// TwinCAT 3 PLC project TestHarnessCoreVerifier
// ProgramVersion: 3.1.4026.24
// libraries:
//   Tc2_Standard, * (Beckhoff Automation GmbH)
//   Tc2_System, * (Beckhoff Automation GmbH)
//   TestHarnessCore, * (None)
// project tree:
//   Doubles/ ConcurrencyWitness.TcPOU, ErroringTest.TcPOU, FailingTest.TcPOU, FakeTest.TcPOU, FakeTestWithAllHooks.TcPOU, FakeTestWithSetup.TcPOU, FloorTest.TcPOU, HangingBodyTest.TcPOU, HangingSetupTest.TcPOU, HangingTeardownTest.TcPOU, OrderedHooksTest.TcPOU, OrderWitness.TcPOU, PassingTest.TcPOU, RecordingReporter.TcPOU, SetupFailsTest.TcPOU, SlowSetupTest.TcPOU, SpanningTest.TcPOU, SpyReporter.TcPOU, StallingSuite.TcPOU, VerdictOnlyReporter.TcPOU, WitnessedTest.TcPOU
//   DUTs/ E_FloorStage.TcDUT, E_PureColour.TcDUT, ST_PureSample.TcDUT, ST_RecordedCase.TcDUT
//   Interfaces/ I_ProbeWitness.TcIO
//   / PlcTask.TcTTO
//   POUs/ MAIN.TcPOU, PRG_FloorCheck.TcPOU, PRG_UnitTests.TcPOU
//   Tests/Arbiter/ TEST_ArbiterAbandonEndsThePass.TcPOU, TEST_ArbiterCurrentIsNullWhenNothingActive.TcPOU, TEST_ArbiterEmptyPassIsComplete.TcPOU, TEST_ArbiterNotExhaustedWhileLastTestRuns.TcPOU, TEST_ArbiterRestartsFromTheBeginning.TcPOU, TEST_ArbiterVisitsEveryTestOnce.TcPOU
//   Tests/Assertions/ TEST_AssertBufferComparisons.TcPOU, TEST_AssertCompletedWithinCountsCompletedScans.TcPOU, TEST_AssertGreaterAndLessCompareTheRightWayRound.TcPOU, TEST_AssertInRangeIsInclusive.TcPOU, TEST_AssertNearUsesAbsoluteTolerance.TcPOU, TEST_AssertNotEqualRejectsSameness.TcPOU, TEST_AssertWithinUsesRelativeTolerance.TcPOU
//   Tests/Characterization/ CHAR_Capacity.TcPOU, CHAR_OverflowStatistics.TcPOU, CHAR_ReRunIndividual.TcPOU, CHAR_ReRunTests.TcPOU, CHAR_SerialExecution.TcPOU, CHAR_TimeoutPrecedence.TcPOU, CHAR_WallClockTimeout.TcPOU
//   Tests/EventReporter/ TEST_EventReporterDoesNotCallASkipAPass.TcPOU, TEST_EventReporterIsQuietAboutPasses.TcPOU, TEST_EventReporterNamesASkippedAndAnErroredRun.TcPOU, TEST_EventReporterRaisesEachOutcomeOnce.TcPOU, TEST_EventReporterSendsAndDoesNotFail.TcPOU, TEST_EventReporterWorksThroughTheFanout.TcPOU
//   Tests/Fanout/ TEST_FanoutCarriesTheSuiteResultThrough.TcPOU, TEST_FanoutForwardsRunStarted.TcPOU, TEST_FanoutIsIdleIsTheAndOfEverySink.TcPOU, TEST_FanoutNotifiesEverySinkInOrder.TcPOU, TEST_FanoutOnlyChecksGoToDetailSinks.TcPOU, TEST_FanoutRefusesBeyondCapacityAndTellsTheRest.TcPOU, TEST_FanoutSuspendSilencesEverything.TcPOU
//   Tests/Journal/ TEST_JournalDefaultsFillOnlyWhatWasNotClaimed.TcPOU, TEST_JournalResetKeepsWhatWasRegistered.TcPOU, TEST_JournalSkippedIsTerminalAndNotRed.TcPOU, TEST_JournalTimesOutOnCycles.TcPOU, TEST_JournalZeroBudgetDisablesTheDeadline.TcPOU
//   Tests/JUnitReporter/ TEST_JUnitReporterIsBusyWhileWriting.TcPOU, TEST_JUnitReporterOpensOnRunStarted.TcPOU, TEST_JUnitReporterRefusesWithNoPath.TcPOU, TEST_JUnitReporterReportsAFailedWrite.TcPOU, TEST_JUnitReporterWritesNothingWhenNothingRan.TcPOU, TEST_JUnitReporterWritesTheDocument.TcPOU
//   Tests/LogReporter/ TEST_LogReporterAlwaysWritesFrameworkErrors.TcPOU, TEST_LogReporterIsQuietAboutPasses.TcPOU, TEST_LogReporterNamesASkippedAndAnErroredRun.TcPOU, TEST_LogReporterNarratesSkipsOnlyWhenAsked.TcPOU, TEST_LogReporterNarratesWhenAsked.TcPOU, TEST_LogReporterSummarisesASuite.TcPOU, TEST_LogReporterWritesFailuresAndErrors.TcPOU
//   Tests/PureFunctions/ TEST_CompareNumericRules.TcPOU, TEST_CompareOtherRules.TcPOU, TEST_CompareTextRules.TcPOU, TEST_StopwatchMeasuresAndFreezes.TcPOU, TEST_SummaryLineComposition.TcPOU, TEST_ValueBriefShortens.TcPOU, TEST_ValueRendering.TcPOU
//   Tests/Registry/ TEST_RegistryCapacityAndOverflow.TcPOU, TEST_RegistryClosesRegistration.TcPOU, TEST_RegistryJournalRejectsBadIndex.TcPOU, TEST_RegistryJournalsArePerSlot.TcPOU, TEST_RegistryLookup.TcPOU, TEST_RegistryPreservesOrder.TcPOU, TEST_RegistryRejectsDuplicateLabel.TcPOU, TEST_RegistryRejectsEmptyLabelAndNullTest.TcPOU, TEST_RegistryResolvesOptionalHooks.TcPOU, TEST_RegistrySlotCarriesItsIndex.TcPOU
//   Tests/Runner/ TEST_RunnerAbandonMakesOneFinalCall.TcPOU, TEST_RunnerBodyDeadlineFires.TcPOU, TEST_RunnerDrivesThePhasesInOrder.TcPOU, TEST_RunnerRefusesAnEmptySlot.TcPOU, TEST_RunnerRunsAMultiScanBody.TcPOU, TEST_RunnerSetupDeadlineFires.TcPOU, TEST_RunnerSetupDoesNotSpendTheBodyBudget.TcPOU, TEST_RunnerSetupFailureSkipsTheBody.TcPOU, TEST_RunnerTeardownOverrunKeepsTheVerdict.TcPOU
//   Tests/Suite/ TEST_RegisteredAndReporterCountsAreReadable.TcPOU, TEST_RunAnnouncesItselfBeforeAnythingElse.TcPOU, TEST_RunOfOnlySkippedTestsIsSkipped.TcPOU, TEST_RunPassesWithSkipsBesideAPass.TcPOU, TEST_RunRefusingASuiteIsNeverSilent.TcPOU, TEST_RunReportsASkippedSuiteInItsPlace.TcPOU, TEST_RunReportsASuiteSkippedBeforeItsReporters.TcPOU, TEST_RunReportsEachSkippedTestByName.TcPOU, TEST_RunReRunDoesNotRunASkippedSuite.TcPOU, TEST_RunReRunReportsASkippedSuiteAgain.TcPOU, TEST_RunWithMoreSkipsThanPassesIsPassed.TcPOU, TEST_SuiteClosesRegistrationOnFirstEnable.TcPOU, TEST_SuiteDefaultsReachTheTests.TcPOU, TEST_SuiteRejectedRegistrationIsNeverSilent.TcPOU, TEST_SuiteReRunRepeatsTheRegisteredSet.TcPOU, TEST_SuiteReRunSingleRecordsNothing.TcPOU, TEST_SuiteRunsEveryRegisteredTest.TcPOU, TEST_SuiteSeparatesFailuresFromErrors.TcPOU, TEST_SuiteSkipMarksEverythingSkipped.TcPOU, TEST_SuiteSkippedAfterARejectedRegistrationIsErrored.TcPOU, TEST_SuiteSkippedWithNoLabelIsAFrameworkError.TcPOU, TEST_SuiteWithNoLabelIsAFrameworkError.TcPOU, TEST_SuiteWithNothingRegisteredIsComplete.TcPOU
//   Tests/Verdict/ TEST_VerdictFailIsAPlainFailure.TcPOU, TEST_VerdictFirstFailureWinsTheSummary.TcPOU, TEST_VerdictPassDoesNotOvertakeAFailure.TcPOU, TEST_VerdictRecordsAFailure.TcPOU, TEST_VerdictReportErrorIsNotAFailure.TcPOU, TEST_VerdictSummaryLeadsWithTheStepLabel.TcPOU, TEST_VerdictUntargetedHandleIsInert.TcPOU, TEST_VerdictZeroChecksIsErrored.TcPOU
//   Tests/Watchdog/ TEST_WatchdogAbandonsAStalledSuite.TcPOU, TEST_WatchdogMeasuresProgressNotTime.TcPOU, TEST_WatchdogZeroDisablesIt.TcPOU
// (motion and I/O tree: see PLC project testharnesscore)
// real-time tasks:
//   TASK PlcTask: cycle T#10ms, priority 20, ADS port 350

CONFIGURATION TestHarnessCoreVerifier
    RESOURCE PLC ON TwinCAT3
        TASK PlcTask(INTERVAL := T#10ms, PRIORITY := 20);
        PROGRAM MAIN WITH PlcTask : MAIN;
    END_RESOURCE
END_CONFIGURATION

// ---- DUTs/E_FloorStage.TcDUT
// Where the floor check has got to. One step per scan, so each stage's effect can

// be seen before the next runs.
{attribute 'qualified_only'}
{attribute 'strict'}
TYPE E_FloorStage : (
		Register := 0,
		Select	 := 1,
		Drive	 := 2,
		Read	 := 3,
		Done	 := 4
	) DINT;
END_TYPE

// ---- DUTs/E_PureColour.TcDUT
// A sample enum, for pinning that enums compare and render at all. The original

// rendered an unrecognised type class as an empty string, so a failed enum

// comparison read 'expected , actual ' - nothing, at the moment the reader most

// needed something.
{attribute 'qualified_only'}
TYPE E_PureColour : (
		Red	  := 0,
		Green := 1,
		Blue  := 2
	) DINT;
END_TYPE

// ---- DUTs/ST_PureSample.TcDUT
// A sample record for comparison tests. Shaped like a CoE object entry because

// that is the kind of struct a real test compares.
TYPE ST_PureSample :
	STRUCT
		Index	 : WORD;
		SubIndex : BYTE;
		Value	 : DINT;
	END_STRUCT
END_TYPE

// ---- DUTs/ST_RecordedCase.TcDUT
// One testcase as a recording sink captured it - the in-memory equivalent of a

// <testcase> node in the result document.

//

// The characterization tests ask questions of the ARTIFACT, not of the counters:

// how many cases, what failure type, does the message name the wall clock. This

// is what lets them, without a file to read back.
TYPE ST_RecordedCase :
	STRUCT
		Label	 : T_MaxString;
		Location : T_MaxString;
		Status	 : E_TestStatus;
		Kind	 : E_FailureKind;
		Summary	 : T_MaxString;
	END_STRUCT
END_TYPE

// ---- Interfaces/I_ProbeWitness.TcIO
// Somewhere for several spies to record the order they were notified in.

//

// An interface rather than a shared instance, because a spy holding the concrete

// type would be a second thing to keep wired up correctly.
INTERFACE I_ProbeWitness EXTENDS __SYSTEM.IQueryInterface

// Called by each spy as it is notified. Ordinal identifies which one.
METHOD Note
VAR_INPUT
	Ordinal : UDINT;
END_VAR
END_METHOD

END_INTERFACE

// ---- POUs/MAIN.TcPOU
// The verifier's task entry point.

//

// The floor check stands alone and runs first: it proves the harness can run a

// test at all, WITHOUT using the harness to prove it. Read PRG_FloorCheck.AllGood

// before trusting anything in PRG_UnitTests - if the runner is broken, every test

// reports NotStarted and that looks exactly like a wiring mistake.
PROGRAM MAIN

PRG_FloorCheck();
PRG_UnitTests();

END_PROGRAM

// ---- POUs/PRG_FloorCheck.TcPOU
// Proves the harness can run one test and report a verdict - WITHOUT using the

// harness to prove it.

//

// The verifier tests TestHarnessCore using TestHarnessCore. That is unavoidable

// and mostly fine, but it leaves one hole: if the runner never advances, every

// test reports NotStarted, and that looks exactly like a wiring mistake. There is

// no way to tell a framework defect from a setup error, because the thing

// reporting the result is the thing under test.

//

// So this drives TestRegistry, TestArbiter and TestRunner BY HAND, one step per

// scan, and writes what it finds into plain variables. Read them in the online

// view. Nothing between you and those objects is itself under test.

//

// EXPECTED once Stage reaches Done:

//

//   Claimed        TRUE          Advanced       TRUE

//   ActiveLabel    'floor'       Loaded         TRUE

//   Outcome        Finished      Verdict        Passed

//   Checks         1             BodyRunCount   1

//   Exhausted      TRUE          AllGood        TRUE

//

// AllGood is every line above, ANDed. If it is TRUE the floor holds, and any

// failure a real test reports afterwards is a real finding.

//

// If it is FALSE, read the values individually: the first wrong one names the

// object that broke.

//

// Re-run after ANY change to TestRunner, TestArbiter or TestRegistry. It costs one

// scan and it is the only check here that does not depend on what it tests.
PROGRAM PRG_FloorCheck
VAR
	// -- driven directly, not through a suite -----------------------------------
	Registry : TestRegistry<2>;
	Arbiter	 : TestArbiter;
	Runner	 : TestRunner;

	// The assertion handle. Named Handle, not Verdict, so it cannot be confused

	// with the verdict the test earns.
	Handle	: TestVerdict;
	Subject : FloorTest;
	Budgets : ST_TestBudgets;

	// -- what was found ---------------------------------------------------------
	Stage		 : E_FloorStage;
	Claimed		 : BOOL;
	Advanced	 : BOOL;
	ActiveLabel	 : T_MaxString;
	Loaded		 : BOOL;
	Outcome		 : E_PhaseOutcome;
	Verdict		 : E_TestStatus;
	Checks		 : UDINT;
	BodyRunCount : UDINT;
	Exhausted	 : BOOL;
	AllGood		 : BOOL;

	// -- working ----------------------------------------------------------------
	Slot	: ST_TestSlot;
	Journal : REFERENCE TO TestJournal;
	Fault	: E_RegistrationFault;
END_VAR

CASE Stage OF
	E_FloorStage.Register:
		// Capacity 2 holding one test. Capacity is not what is being checked here.
		Fault	:= Registry.TryClaim(Subject, 'floor', Budgets);
		Claimed := (Fault = E_RegistrationFault.None);
		Runner.Attach(Roster := Registry, Verdict := Handle);
		Arbiter.Attach(Registry);
		Arbiter.Begin();
		Stage := E_FloorStage.Select;

	E_FloorStage.Select:
		Advanced	:= Arbiter.Advance();
		Slot		:= Arbiter.Current;
		ActiveLabel := Slot.Label;
		Loaded		:= Runner.Load(Slot);
		Stage		:= E_FloorStage.Drive;

	E_FloorStage.Drive:
		// One scan of the body. A single-scan test must finish here; if it does not,
		// Outcome stays Running and that is itself the finding.
		Outcome := Runner.Advance(Enable := TRUE);
		IF Outcome <> E_PhaseOutcome.Running THEN
			Stage := E_FloorStage.Read;
		END_IF

	E_FloorStage.Read:
		Journal REF= Registry.Journal(0);
		IF __ISVALIDREF(Journal) THEN
			Verdict := Journal.Status;
			Checks	:= Journal.AssertionCount;
		END_IF

		BodyRunCount := Subject.RunCount;

		// Nothing left to hand out and nothing running.
		Arbiter.Advance();
		Exhausted := Arbiter.IsExhausted;
		AllGood	  := Claimed AND Advanced AND (ActiveLabel = 'floor') AND Loaded AND (Outcome = E_PhaseOutcome.Finished) AND (Verdict = E_TestStatus.Passed) AND (Checks = 1) AND (BodyRunCount = 1) AND Exhausted;
		Stage	  := E_FloorStage.Done;

	E_FloorStage.Done:
		// Terminal. Nothing repeats, so every value above stays readable.
		;
END_CASE

END_PROGRAM

// ---- Doubles/FloorTest.TcPOU
// The simplest thing that can be called a test: one check, finished in one scan.

//

// Nothing optional, nothing multi-scan, nothing that can fail. If the harness

// cannot run THIS and report Passed, no other result it produces means anything.
FUNCTION_BLOCK FloorTest IMPLEMENTS I_Test
VAR
	// Counted so the floor check can prove the body ran exactly once. A harness

	// that called it twice, or never, would otherwise look identical from outside.
	_RunCount : UDINT;
END_VAR

METHOD Run : BOOL
VAR_INPUT
	Enable : BOOL;
	Test   : I_TestAssertions;
END_VAR

VAR
	// AssertEqual takes ANY, which binds only to an addressable variable - a

	// literal or an inlined expression will not compile. Both sides are copied into

	// variables first. A language constraint, not a choice.
	Expected : DINT := 4;
	Actual	 : DINT;
	Two		 : DINT := 2;
END_VAR
IF NOT Enable THEN
	// Abandoned. Nothing to unwind.
	Run := TRUE;
	RETURN;
END_IF

_RunCount := _RunCount + 1;
Actual	  := Two + Two;
Test.AssertEqual(Expected, Actual, 'two and two');
Run := TRUE;
END_METHOD

// How many times the harness called Run. Exactly 1 after a clean single run.
PROPERTY RunCount : UDINT
GET
RunCount := _RunCount;
END_GET
END_PROPERTY

END_FUNCTION_BLOCK

// ---- POUs/PRG_UnitTests.TcPOU
// The composition root: what is registered, what reports it, and the run that
// drives it.
//
// This is also a WORKED EXAMPLE. It composes the library the way a real project
// should - a run, a suite, three sinks - so anything awkward here is awkward for
// everyone.
//
// READ THESE, in the online view:
//
//   Complete   TRUE once every test has finished
//   Outcome    Passed if the library is sound
//   Total      111 - assert this. A test that stops being registered vanishes
//              silently, and CI sees fewer passes rather than a failure
//   Passed / Failed / Errors / Skipped
//   Idle       TRUE once the result document has reached disk. CI MUST WAIT FOR
//              BOTH Complete AND Idle - a run finishing and its file landing are
//              different events, and copying between them yields a truncated
//              artifact that reads as a broken pipeline
//
// WHERE A FAILURE SHOWS UP:
//   - the Logged Events window, as a log line and as an event
//   - C:\ProgramData\Beckhoff\TwinCAT\3.1\Boot\TestHarnessCoreResults.xml
//
// Read the failure there rather than from journal internals in a watch window.
// Making that unnecessary is what this library is for.
//
// THE FAILURE PATH IS EXERCISED, not assumed. The Verdict tests drive DELIBERATE
// failures into a private journal; the Suite tests register doubles that fail and
// error on purpose; the JUnit tests write to a folder that does not exist. They all
// pass. What they prove is that going wrong works.
//
// THE CHARACTERIZATION TESTS ARE THE ACCEPTANCE CONTRACT - behaviour a project
// depending on this library is entitled to rely on. They are also the only tests
// that ask questions of the ARTIFACT: how many cases the document carries, what
// type attribute a failure got, whether a timeout message names the wall clock.
//
// MULTI-SCAN TESTS hold a private runner, suite or run and step it one scan per
// call, returning FALSE until it finishes - the same mechanism they are verifying,
// one level down. Each carries a watchdog, so a defect that never completes fails
// its own test rather than hanging everything and looking like a broken verifier.
PROGRAM PRG_UnitTests
VAR
	// A RUN, not just a suite. RunFinished is a run-level event and only a TestRun
	// raises it - which is what produces a document at all.
	Runner : TestRun<2>;
	Suite  : TestSuite<130>;

	// All three sinks, which is the realistic composition: a log line to read at a
	// glance, an event to filter and route, a document for CI.
	LogSink	  : TestLogReporter;
	EventSink : TestEventReporter;
	JUnitSink : TestJUnitReporter;

	// The 4026 boot folder. Named apart from the files the JUnit tests write, so a
	// stale artifact from either cannot be mistaken for the other.
	ResultPath : T_MaxString := 'C:\ProgramData\Beckhoff\TwinCAT\3.1\Boot\TestHarnessCoreResults.xml';

	Budgets : ST_TestBudgets;
	Wired	: BOOL;

	// -- Registry --
	registryCapacityAndOverflow	: TEST_RegistryCapacityAndOverflow;
	registryRejectsDuplicateLabel	: TEST_RegistryRejectsDuplicateLabel;
	registryRejectsEmptyLabelAndNullTest	: TEST_RegistryRejectsEmptyLabelAndNullTest;
	registryClosesRegistration	: TEST_RegistryClosesRegistration;
	registryLookup	: TEST_RegistryLookup;
	registryPreservesOrder	: TEST_RegistryPreservesOrder;
	registrySlotCarriesItsIndex	: TEST_RegistrySlotCarriesItsIndex;
	registryResolvesOptionalHooks	: TEST_RegistryResolvesOptionalHooks;
	registryJournalsArePerSlot	: TEST_RegistryJournalsArePerSlot;
	registryJournalRejectsBadIndex	: TEST_RegistryJournalRejectsBadIndex;

	// -- Arbiter --
	arbiterVisitsEveryTestOnce	: TEST_ArbiterVisitsEveryTestOnce;
	arbiterCurrentIsNullWhenNothingActive	: TEST_ArbiterCurrentIsNullWhenNothingActive;
	arbiterEmptyPassIsComplete	: TEST_ArbiterEmptyPassIsComplete;
	arbiterAbandonEndsThePass	: TEST_ArbiterAbandonEndsThePass;
	arbiterNotExhaustedWhileLastTestRuns	: TEST_ArbiterNotExhaustedWhileLastTestRuns;
	arbiterRestartsFromTheBeginning	: TEST_ArbiterRestartsFromTheBeginning;

	// -- Verdict --
	verdictRecordsAFailure	: TEST_VerdictRecordsAFailure;
	verdictPassDoesNotOvertakeAFailure	: TEST_VerdictPassDoesNotOvertakeAFailure;
	verdictZeroChecksIsErrored	: TEST_VerdictZeroChecksIsErrored;
	verdictReportErrorIsNotAFailure	: TEST_VerdictReportErrorIsNotAFailure;
	verdictFailIsAPlainFailure	: TEST_VerdictFailIsAPlainFailure;
	verdictSummaryLeadsWithTheStepLabel	: TEST_VerdictSummaryLeadsWithTheStepLabel;
	verdictFirstFailureWinsTheSummary	: TEST_VerdictFirstFailureWinsTheSummary;
	verdictUntargetedHandleIsInert	: TEST_VerdictUntargetedHandleIsInert;

	// -- Journal --
	journalTimesOutOnCycles	: TEST_JournalTimesOutOnCycles;
	journalZeroBudgetDisablesTheDeadline	: TEST_JournalZeroBudgetDisablesTheDeadline;
	journalDefaultsFillOnlyWhatWasNotClaimed	: TEST_JournalDefaultsFillOnlyWhatWasNotClaimed;
	journalResetKeepsWhatWasRegistered	: TEST_JournalResetKeepsWhatWasRegistered;
	journalSkippedIsTerminalAndNotRed	: TEST_JournalSkippedIsTerminalAndNotRed;

	// -- Runner --
	runnerDrivesThePhasesInOrder	: TEST_RunnerDrivesThePhasesInOrder;
	runnerRunsAMultiScanBody	: TEST_RunnerRunsAMultiScanBody;
	runnerSetupFailureSkipsTheBody	: TEST_RunnerSetupFailureSkipsTheBody;
	runnerSetupDoesNotSpendTheBodyBudget	: TEST_RunnerSetupDoesNotSpendTheBodyBudget;
	runnerBodyDeadlineFires	: TEST_RunnerBodyDeadlineFires;
	runnerSetupDeadlineFires	: TEST_RunnerSetupDeadlineFires;
	runnerTeardownOverrunKeepsTheVerdict	: TEST_RunnerTeardownOverrunKeepsTheVerdict;
	runnerAbandonMakesOneFinalCall	: TEST_RunnerAbandonMakesOneFinalCall;
	runnerRefusesAnEmptySlot	: TEST_RunnerRefusesAnEmptySlot;

	// -- Suite --
	suiteRunsEveryRegisteredTest	: TEST_SuiteRunsEveryRegisteredTest;
	suiteSeparatesFailuresFromErrors	: TEST_SuiteSeparatesFailuresFromErrors;
	suiteClosesRegistrationOnFirstEnable	: TEST_SuiteClosesRegistrationOnFirstEnable;
	suiteRejectedRegistrationIsNeverSilent	: TEST_SuiteRejectedRegistrationIsNeverSilent;
	suiteSkipMarksEverythingSkipped	: TEST_SuiteSkipMarksEverythingSkipped;
	suiteSkippedAfterARejectedRegistrationIsErrored	: TEST_SuiteSkippedAfterARejectedRegistrationIsErrored;
	suiteSkippedWithNoLabelIsAFrameworkError	: TEST_SuiteSkippedWithNoLabelIsAFrameworkError;
	suiteReRunRepeatsTheRegisteredSet	: TEST_SuiteReRunRepeatsTheRegisteredSet;
	suiteReRunSingleRecordsNothing	: TEST_SuiteReRunSingleRecordsNothing;
	suiteWithNothingRegisteredIsComplete	: TEST_SuiteWithNothingRegisteredIsComplete;
	suiteWithNoLabelIsAFrameworkError	: TEST_SuiteWithNoLabelIsAFrameworkError;
	suiteDefaultsReachTheTests	: TEST_SuiteDefaultsReachTheTests;

	runAnnouncesItselfBeforeAnythingElse	: TEST_RunAnnouncesItselfBeforeAnythingElse;
	runRefusingASuiteIsNeverSilent	: TEST_RunRefusingASuiteIsNeverSilent;
	runPassesWithSkipsBesideAPass	: TEST_RunPassesWithSkipsBesideAPass;
	runOfOnlySkippedTestsIsSkipped	: TEST_RunOfOnlySkippedTestsIsSkipped;
	runWithMoreSkipsThanPassesIsPassed	: TEST_RunWithMoreSkipsThanPassesIsPassed;
	runReportsASuiteSkippedBeforeItsReporters	: TEST_RunReportsASuiteSkippedBeforeItsReporters;
	runReportsASkippedSuiteInItsPlace	: TEST_RunReportsASkippedSuiteInItsPlace;
	runReportsEachSkippedTestByName	: TEST_RunReportsEachSkippedTestByName;
	runReRunDoesNotRunASkippedSuite	: TEST_RunReRunDoesNotRunASkippedSuite;
	runReRunReportsASkippedSuiteAgain	: TEST_RunReRunReportsASkippedSuiteAgain;

	// -- Fanout --
	fanoutNotifiesEverySinkInOrder	: TEST_FanoutNotifiesEverySinkInOrder;
	fanoutOnlyChecksGoToDetailSinks	: TEST_FanoutOnlyChecksGoToDetailSinks;
	fanoutIsIdleIsTheAndOfEverySink	: TEST_FanoutIsIdleIsTheAndOfEverySink;
	fanoutSuspendSilencesEverything	: TEST_FanoutSuspendSilencesEverything;
	fanoutRefusesBeyondCapacityAndTellsTheRest	: TEST_FanoutRefusesBeyondCapacityAndTellsTheRest;
	fanoutCarriesTheSuiteResultThrough	: TEST_FanoutCarriesTheSuiteResultThrough;

	fanoutForwardsRunStarted	: TEST_FanoutForwardsRunStarted;

	// -- LogReporter --
	logReporterIsQuietAboutPasses	: TEST_LogReporterIsQuietAboutPasses;
	logReporterWritesFailuresAndErrors	: TEST_LogReporterWritesFailuresAndErrors;
	logReporterNarratesWhenAsked	: TEST_LogReporterNarratesWhenAsked;
	logReporterAlwaysWritesFrameworkErrors	: TEST_LogReporterAlwaysWritesFrameworkErrors;
	logReporterSummarisesASuite	: TEST_LogReporterSummarisesASuite;
	logReporterNarratesSkipsOnlyWhenAsked	: TEST_LogReporterNarratesSkipsOnlyWhenAsked;
	logReporterNamesASkippedAndAnErroredRun	: TEST_LogReporterNamesASkippedAndAnErroredRun;

	jUnitReporterOpensOnRunStarted	: TEST_JUnitReporterOpensOnRunStarted;

	// -- EventReporter --
	eventReporterSendsAndDoesNotFail	: TEST_EventReporterSendsAndDoesNotFail;
	eventReporterIsQuietAboutPasses	: TEST_EventReporterIsQuietAboutPasses;
	eventReporterRaisesEachOutcomeOnce	: TEST_EventReporterRaisesEachOutcomeOnce;
	eventReporterWorksThroughTheFanout	: TEST_EventReporterWorksThroughTheFanout;
	eventReporterDoesNotCallASkipAPass	: TEST_EventReporterDoesNotCallASkipAPass;
	eventReporterNamesASkippedAndAnErroredRun	: TEST_EventReporterNamesASkippedAndAnErroredRun;

	// -- JUnitReporter --
	jUnitReporterWritesTheDocument	: TEST_JUnitReporterWritesTheDocument;
	jUnitReporterIsBusyWhileWriting	: TEST_JUnitReporterIsBusyWhileWriting;
	jUnitReporterReportsAFailedWrite	: TEST_JUnitReporterReportsAFailedWrite;
	jUnitReporterRefusesWithNoPath	: TEST_JUnitReporterRefusesWithNoPath;
	jUnitReporterWritesNothingWhenNothingRan	: TEST_JUnitReporterWritesNothingWhenNothingRan;

	// -- Pure functions: the comparison and rendering rules --
	compareNumericRules	: TEST_CompareNumericRules;
	compareTextRules	: TEST_CompareTextRules;
	compareOtherRules	: TEST_CompareOtherRules;
	summaryLineComposition	: TEST_SummaryLineComposition;
	valueRendering	: TEST_ValueRendering;
	valueBriefShortens	: TEST_ValueBriefShortens;

	// -- Assertions: the public surface every user touches --
	assertNotEqualRejectsSameness	: TEST_AssertNotEqualRejectsSameness;
	assertGreaterAndLessCompareTheRightWayRound	: TEST_AssertGreaterAndLessCompareTheRightWayRound;
	assertNearUsesAbsoluteTolerance	: TEST_AssertNearUsesAbsoluteTolerance;
	assertWithinUsesRelativeTolerance	: TEST_AssertWithinUsesRelativeTolerance;
	assertInRangeIsInclusive	: TEST_AssertInRangeIsInclusive;
	assertBufferComparisons	: TEST_AssertBufferComparisons;
	assertCompletedWithinCountsCompletedScans	: TEST_AssertCompletedWithinCountsCompletedScans;

	stopwatchMeasuresAndFreezes	: TEST_StopwatchMeasuresAndFreezes;
	registeredAndReporterCountsAreReadable	: TEST_RegisteredAndReporterCountsAreReadable;
	// -- Suite watchdog --
	watchdogAbandonsAStalledSuite	: TEST_WatchdogAbandonsAStalledSuite;
	watchdogMeasuresProgressNotTime	: TEST_WatchdogMeasuresProgressNotTime;
	watchdogZeroDisablesIt	: TEST_WatchdogZeroDisablesIt;

	// -- Characterization: the acceptance contract --
	cHAR_Capacity	: CHAR_Capacity;
	cHAR_OverflowStatistics	: CHAR_OverflowStatistics;
	cHAR_ReRunTests	: CHAR_ReRunTests;
	cHAR_ReRunIndividual	: CHAR_ReRunIndividual;
	cHAR_WallClockTimeout	: CHAR_WallClockTimeout;
	cHAR_TimeoutPrecedence	: CHAR_TimeoutPrecedence;
	cHAR_SerialExecution	: CHAR_SerialExecution;

	// -- the result, for the watch window ---------------------------------------
	Complete : BOOL;
	Outcome	 : E_RunOutcome;
	Total	 : UDINT;
	Passed	 : UDINT;
	Failed	 : UDINT;
	Errors	 : UDINT;
	Skipped	 : UDINT;
	Duration : LREAL;

	// -- did the artifact land? -------------------------------------------------
	Idle		  : BOOL;
	FilesWritten  : UDINT;
	WriteFailures : UDINT;
END_VAR

IF NOT Wired THEN
	Wired := TRUE;

	Suite.SetLabel('TestHarnessCore');

	// Registry
	Suite.Register(registryCapacityAndOverflow, 'Registry: capacity and overflow', Budgets);
	Suite.Register(registryRejectsDuplicateLabel, 'Registry: rejects a duplicate label', Budgets);
	Suite.Register(registryRejectsEmptyLabelAndNullTest, 'Registry: rejects an empty label and a null test', Budgets);
	Suite.Register(registryClosesRegistration, 'Registry: closes registration on first enable', Budgets);
	Suite.Register(registryLookup, 'Registry: lookup by label', Budgets);
	Suite.Register(registryPreservesOrder, 'Registry: preserves registration order', Budgets);
	Suite.Register(registrySlotCarriesItsIndex, 'Registry: a slot carries its own index', Budgets);
	Suite.Register(registryResolvesOptionalHooks, 'Registry: resolves the optional hooks independently', Budgets);
	Suite.Register(registryJournalsArePerSlot, 'Registry: journals are per slot and live', Budgets);
	Suite.Register(registryJournalRejectsBadIndex, 'Registry: an out-of-range journal is invalid', Budgets);

	// Arbiter
	Suite.Register(arbiterVisitsEveryTestOnce, 'Arbiter: visits every test once, in order', Budgets);
	Suite.Register(arbiterCurrentIsNullWhenNothingActive, 'Arbiter: current is null when nothing is active', Budgets);
	Suite.Register(arbiterEmptyPassIsComplete, 'Arbiter: an empty pass is complete, not stuck', Budgets);
	Suite.Register(arbiterAbandonEndsThePass, 'Arbiter: abandon does not visit the rest', Budgets);
	Suite.Register(arbiterNotExhaustedWhileLastTestRuns, 'Arbiter: not exhausted while the last test runs', Budgets);
	Suite.Register(arbiterRestartsFromTheBeginning, 'Arbiter: begin restarts from the first test', Budgets);

	// Verdict
	Suite.Register(verdictRecordsAFailure, 'Verdict: a mismatched check is recorded as a failure', Budgets);
	Suite.Register(verdictPassDoesNotOvertakeAFailure, 'Verdict: a pass cannot undo a failure', Budgets);
	Suite.Register(verdictZeroChecksIsErrored, 'Verdict: finishing with no checks is Errored', Budgets);
	Suite.Register(verdictReportErrorIsNotAFailure, 'Verdict: ReportError produces Errored, not Failed', Budgets);
	Suite.Register(verdictFailIsAPlainFailure, 'Verdict: Fail produces Failed', Budgets);
	Suite.Register(verdictSummaryLeadsWithTheStepLabel, 'Verdict: the summary leads with the step label', Budgets);
	Suite.Register(verdictFirstFailureWinsTheSummary, 'Verdict: the first failure wins the summary', Budgets);
	Suite.Register(verdictUntargetedHandleIsInert, 'Verdict: an untargeted handle records nothing', Budgets);

	// Journal
	Suite.Register(journalTimesOutOnCycles, 'Journal: a scan budget expires and records itself', Budgets);
	Suite.Register(journalZeroBudgetDisablesTheDeadline, 'Journal: a zero budget never expires', Budgets);
	Suite.Register(journalDefaultsFillOnlyWhatWasNotClaimed, 'Journal: defaults fill only unclaimed units', Budgets);
	Suite.Register(journalResetKeepsWhatWasRegistered, 'Journal: reset clears the verdict, keeps the budgets', Budgets);
	Suite.Register(journalSkippedIsTerminalAndNotRed, 'Journal: skipped is terminal and not a failure', Budgets);

	// Runner
	Suite.Register(runnerDrivesThePhasesInOrder, 'Runner: setup, body, teardown, each once, in order', Budgets);
	Suite.Register(runnerRunsAMultiScanBody, 'Runner: a multi-scan body is called until it finishes', Budgets);
	Suite.Register(runnerSetupFailureSkipsTheBody, 'Runner: a failed setup skips the body but not teardown', Budgets);
	Suite.Register(runnerSetupDoesNotSpendTheBodyBudget, 'Runner: setup does not spend the body scan budget', Budgets);
	Suite.Register(runnerBodyDeadlineFires, 'Runner: the body deadline stops a hanging test', Budgets);
	Suite.Register(runnerSetupDeadlineFires, 'Runner: setup has its own deadline', Budgets);
	Suite.Register(runnerTeardownOverrunKeepsTheVerdict, 'Runner: a teardown overrun does not change the verdict', Budgets);
	Suite.Register(runnerAbandonMakesOneFinalCall, 'Runner: abandon makes one final call and skips teardown', Budgets);
	Suite.Register(runnerRefusesAnEmptySlot, 'Runner: an empty slot is refused', Budgets);

	// Suite
	Suite.Register(suiteRunsEveryRegisteredTest, 'Suite: runs every registered test, once', Budgets);
	Suite.Register(suiteSeparatesFailuresFromErrors, 'Suite: failures and errors are counted apart', Budgets);
	Suite.Register(suiteClosesRegistrationOnFirstEnable, 'Suite: registration closes on first enable', Budgets);
	Suite.Register(suiteRejectedRegistrationIsNeverSilent, 'Suite: a rejected registration is never silent', Budgets);
	Suite.Register(suiteSkipMarksEverythingSkipped, 'Suite: Skip marks everything skipped and completes', Budgets);
	Suite.Register(suiteSkippedAfterARejectedRegistrationIsErrored, 'Suite: a registration refused before a skip is still counted', Budgets);
	Suite.Register(suiteSkippedWithNoLabelIsAFrameworkError, 'Suite: a skipped suite with no label is a framework error', Budgets);
	Suite.Register(suiteReRunRepeatsTheRegisteredSet, 'Suite: a re-run repeats the registered set', Budgets);
	Suite.Register(suiteReRunSingleRecordsNothing, 'Suite: an individual re-run records nothing', Budgets);
	Suite.Register(suiteWithNothingRegisteredIsComplete, 'Suite: an empty suite is complete, not red', Budgets);
	Suite.Register(suiteWithNoLabelIsAFrameworkError, 'Suite: an unnamed suite is a framework error', Budgets);
	Suite.Register(suiteDefaultsReachTheTests, 'Suite: suite defaults reach every unclaimed test', Budgets);

	Suite.Register(runAnnouncesItselfBeforeAnythingElse, 'Suite: a run announces itself before any result in it', Budgets);
	Suite.Register(runRefusingASuiteIsNeverSilent, 'Suite: a suite refused at composition still turns the run red', Budgets);
	Suite.Register(runPassesWithSkipsBesideAPass, 'Suite: a run with a pass and skips beside it is Passed', Budgets);
	Suite.Register(runOfOnlySkippedTestsIsSkipped, 'Suite: a run in which every test was skipped is Skipped', Budgets);
	Suite.Register(runWithMoreSkipsThanPassesIsPassed, 'Suite: a run with more skips than passes is still Passed', Budgets);
	Suite.Register(runReportsASuiteSkippedBeforeItsReporters, 'Suite: a suite skipped before its reporters were attached still reaches them', Budgets);
	Suite.Register(runReportsASkippedSuiteInItsPlace, 'Suite: a skipped suite is reported in its place in the run, not when Skip was called', Budgets);
	Suite.Register(runReportsEachSkippedTestByName, 'Suite: every skipped test reaches the sinks by name, before its suite closes', Budgets);
	Suite.Register(runReRunDoesNotRunASkippedSuite, 'Suite: a re-run does not run the tests of a skipped suite', Budgets);
	Suite.Register(runReRunReportsASkippedSuiteAgain, 'Suite: a re-run reports a skipped suite again, as skipped', Budgets);

	// Fanout
	Suite.Register(fanoutNotifiesEverySinkInOrder, 'Fanout: every sink is notified, in attachment order', Budgets);
	Suite.Register(fanoutOnlyChecksGoToDetailSinks, 'Fanout: only detail sinks receive checks', Budgets);
	Suite.Register(fanoutIsIdleIsTheAndOfEverySink, 'Fanout: IsIdle is the AND of every sink', Budgets);
	Suite.Register(fanoutSuspendSilencesEverything, 'Fanout: Suspend silences notifications but not CyclicLogic', Budgets);
	Suite.Register(fanoutRefusesBeyondCapacityAndTellsTheRest, 'Fanout: attachment beyond capacity is refused and reported', Budgets);
	Suite.Register(fanoutCarriesTheSuiteResultThrough, 'Fanout: SuiteFinished carries the live read model', Budgets);

	Suite.Register(fanoutForwardsRunStarted, 'Fanout: RunStarted reaches every sink and Suspend silences it', Budgets);

	// LogReporter
	Suite.Register(logReporterIsQuietAboutPasses, 'LogReporter: quiet about passes by default', Budgets);
	Suite.Register(logReporterWritesFailuresAndErrors, 'LogReporter: failures and errors are written and counted apart', Budgets);
	Suite.Register(logReporterNarratesWhenAsked, 'LogReporter: verbosity turns narration on and off', Budgets);
	Suite.Register(logReporterAlwaysWritesFrameworkErrors, 'LogReporter: framework errors are never suppressed', Budgets);
	Suite.Register(logReporterSummarisesASuite, 'LogReporter: one line per suite, carrying the counts', Budgets);
	Suite.Register(logReporterNarratesSkipsOnlyWhenAsked, 'LogReporter: a skip is narrated only when asked, and never as a failure', Budgets);
	Suite.Register(logReporterNamesASkippedAndAnErroredRun, 'LogReporter: a skipped run and an errored run each get their own banner', Budgets);

	Suite.Register(jUnitReporterOpensOnRunStarted, 'JUnitReporter: the document opens on RunStarted', Budgets);

	// EventReporter
	Suite.Register(eventReporterSendsAndDoesNotFail, 'EventReporter: an event is accepted and no HRESULT is returned', Budgets);
	Suite.Register(eventReporterIsQuietAboutPasses, 'EventReporter: quiet about passes until narration is asked for', Budgets);
	Suite.Register(eventReporterRaisesEachOutcomeOnce, 'EventReporter: one event per notification, none raised twice', Budgets);
	Suite.Register(eventReporterWorksThroughTheFanout, 'EventReporter: it sits behind the fan-out beside the log sink', Budgets);
	Suite.Register(eventReporterDoesNotCallASkipAPass, 'EventReporter: a skipped test raises no event, and never TestPassed', Budgets);
	Suite.Register(eventReporterNamesASkippedAndAnErroredRun, 'EventReporter: a skipped run and an errored run each raise their own event', Budgets);

	// JUnitReporter
	Suite.Register(jUnitReporterWritesTheDocument, 'JUnitReporter: the document reaches disk', Budgets);
	Suite.Register(jUnitReporterIsBusyWhileWriting, 'JUnitReporter: IsIdle is FALSE until the file lands', Budgets);
	Suite.Register(jUnitReporterReportsAFailedWrite, 'JUnitReporter: a failed write is counted and reported (R3)', Budgets);
	Suite.Register(jUnitReporterRefusesWithNoPath, 'JUnitReporter: no path set is a failure, not silence', Budgets);
	Suite.Register(jUnitReporterWritesNothingWhenNothingRan, 'JUnitReporter: an empty run produces no document', Budgets);

	// Pure functions - what equality and rendering MEAN. The object tests exercise
	// them incidentally, whenever some test happens to call AssertEqual, which is
	// not the same as pinning the rules themselves.
	Suite.Register(compareNumericRules, 'Pure: numeric rules: value across widths, exact floats, the hint', Budgets);
	Suite.Register(compareTextRules, 'Pure: string rules: content not capacity, and WSTRING as WSTRING (R1)', Budgets);
	Suite.Register(compareOtherRules, 'Pure: structs, arrays and enums; a size difference is a type difference', Budgets);
	Suite.Register(summaryLineComposition, 'Pure: composition order; the message is dropped whole, not cut', Budgets);
	Suite.Register(valueRendering, 'Pure: values render as something, including enums', Budgets);
	Suite.Register(valueBriefShortens, 'Pure: long values are shortened and marked', Budgets);

	// Assertions - the part of the library every user touches. Each of these checks
	// the direction that would be silently wrong, not just the happy path: a
	// reversed comparison passes every test written against it.
	Suite.Register(assertNotEqualRejectsSameness, 'Assertion: AssertNotEqual passes on difference, fails on sameness', Budgets);
	Suite.Register(assertGreaterAndLessCompareTheRightWayRound, 'Assertion: ordering runs the way the name says, both directions', Budgets);
	Suite.Register(assertNearUsesAbsoluteTolerance, 'Assertion: an absolute band, inclusive and symmetric', Budgets);
	Suite.Register(assertWithinUsesRelativeTolerance, 'Assertion: a relative band that holds across magnitudes', Budgets);
	Suite.Register(assertInRangeIsInclusive, 'Assertion: inclusive on both bounds', Budgets);
	Suite.Register(assertBufferComparisons, 'Assertion: byte offset, size mismatch, and a null buffer', Budgets);
	Suite.Register(assertCompletedWithinCountsCompletedScans, 'Assertion: the scan in progress is not counted', Budgets);

	Suite.Register(stopwatchMeasuresAndFreezes, 'Pure: the stopwatch advances, freezes and resets', Budgets);
	Suite.Register(registeredAndReporterCountsAreReadable, 'Suite: the counts CI is told to assert are readable', Budgets);
	// Suite watchdog - the run is the only object positioned to see a suite that
	// has stopped, because the suite IS the thing that stopped.
	Suite.Register(watchdogAbandonsAStalledSuite, 'Watchdog: a stalled suite is named, abandoned and counted', Budgets);
	Suite.Register(watchdogMeasuresProgressNotTime, 'Watchdog: a progressing suite is never abandoned, however slow', Budgets);
	Suite.Register(watchdogZeroDisablesIt, 'Watchdog: a zero budget never fires', Budgets);

	// Characterization - the acceptance contract. Behaviour a project depending on
	// this library is entitled to rely on, and the only tests that ask questions of
	// the result document rather than of a counter.
	Suite.Register(cHAR_Capacity, 'Contract: capacity holds what it says; overflow is reported', Budgets);
	Suite.Register(cHAR_OverflowStatistics, 'Contract: errors are counted apart from failures', Budgets);
	Suite.Register(cHAR_ReRunTests, 'Contract: one suite node per run; a re-run produces a fresh document', Budgets);
	Suite.Register(cHAR_ReRunIndividual, 'Contract: an individual re-run records nothing', Budgets);
	Suite.Register(cHAR_WallClockTimeout, 'Contract: the wall-clock deadline fires and names itself', Budgets);
	Suite.Register(cHAR_TimeoutPrecedence, 'Contract: suite default, per-test override, per-unit tracking', Budgets);
	Suite.Register(cHAR_SerialExecution, 'Contract: no test body runs while another is running', Budgets);

	// -- reporting -------------------------------------------------------------
	JUnitSink.SetPath(ResultPath);
	// Where a failed write is reported. Deliberately the log sink and not the
	// fan-out, which would call back into the writer that just failed.
	JUnitSink.AttachErrorSink(LogSink);

	Runner.SetLabel('TestHarnessCoreVerifier');
	// Which BUILD of the library ran, printed in both run banners and written to the
	// result document. The library is resolved as 'newest installed', so the build
	// under test is otherwise invisible. A version names an install, not its
	// contents: bump it for every build that needs telling apart, or two different
	// builds will print the same line.
	Runner.SetTargetInfo(CONCAT('TestHarnessCoreVerifier, library ',
								 TestHarnessCore.stLibVersion_TestHarnessCore.sVersion));

	// Attached to the RUN, which pushes each one into every suite. One attachment
	// point, whatever order suites and sinks are added in.
	Runner.AddReporter(LogSink);
	Runner.AddReporter(EventSink);
	Runner.AddReporter(JUnitSink);

	Runner.AddSuite(Suite);
END_IF

Runner.Run(Enable := TRUE);

// Read from the RUN, not the suite: it is the top of the nest, and the figures
// mean the same thing at every level.
Complete := Runner.IsComplete;
Outcome	 := Runner.Outcome;
Total	 := Runner.TestCount;
Passed	 := Runner.PassedCount;
Failed	 := Runner.FailedCount;
Errors	 := Runner.ErrorCount;
Skipped	 := Runner.SkippedCount;
Duration := Runner.TotalDuration;

Idle		  := JUnitSink.IsIdle;
FilesWritten  := JUnitSink.FilesWritten;
WriteFailures := JUnitSink.WriteFailures;

END_PROGRAM

// ---- Tests/Registry/TEST_RegistryCapacityAndOverflow.TcPOU
// A registry declared with three slots holds three, and the fourth is refused as

// Full rather than accepted or written past the end.

//

// Declaring ARRAY[0..Capacity] rather than ARRAY[0..Capacity - 1] would make a

// suite asked for two hold three, and report a limit of two while holding them.
FUNCTION_BLOCK TEST_RegistryCapacityAndOverflow IMPLEMENTS I_Test
VAR
	Registry	  : TestRegistry<3>;
	Fakes		  : ARRAY[0..3] OF FakeTest;
	Budgets		  : ST_TestBudgets;
	i			  : DINT;
	ExpectedFault : E_RegistrationFault;
	ActualFault	  : E_RegistrationFault;
	ExpectedCount : UDINT;
	ActualCount	  : UDINT;
END_VAR

METHOD Run : BOOL
VAR_INPUT
	Enable : BOOL;
	Test   : I_TestAssertions;
END_VAR
FOR i := 0 TO 2 DO
	ActualFault	  := Registry.TryClaim(Fakes[i], CONCAT('Test ', DINT_TO_STRING(i)), Budgets);
	ExpectedFault := E_RegistrationFault.None;
	Test.AssertEqual(ExpectedFault, ActualFault, 'three slots accepted');
END_FOR

ExpectedCount := 3;
ActualCount	  := Registry.Count;
Test.AssertEqual(ExpectedCount, ActualCount, 'count after filling');
ActualFault	  := Registry.TryClaim(Fakes[3], 'One too many', Budgets);
ExpectedFault := E_RegistrationFault.Full;
Test.AssertEqual(ExpectedFault, ActualFault, 'fourth refused as Full');
ExpectedCount := 3;
ActualCount	  := Registry.Count;
Test.AssertEqual(ExpectedCount, ActualCount, 'count unchanged by refusal');
Run := TRUE;
END_METHOD

END_FUNCTION_BLOCK

// ---- Doubles/FakeTest.TcPOU
// A test that implements I_Test and nothing else.

//

// The null case for hook resolution: Setup, Teardown and Location must all come

// back null for this one.
FUNCTION_BLOCK FakeTest IMPLEMENTS I_Test
VAR
	_RunCount : UDINT;
END_VAR

METHOD Run : BOOL
VAR_INPUT
	Enable : BOOL;
	Test   : I_TestAssertions;
END_VAR
_RunCount := _RunCount + 1;
Run		  := TRUE;
END_METHOD

// Should stay 0 in registry and arbiter tests: neither object calls a test.
PROPERTY RunCount : UDINT
GET
RunCount := _RunCount;
END_GET
END_PROPERTY

END_FUNCTION_BLOCK

// ---- Tests/Registry/TEST_RegistryRejectsDuplicateLabel.TcPOU
// Labels are the key CI trend history is built on, so two tests cannot share one.

// The second claim is refused and takes no slot.
FUNCTION_BLOCK TEST_RegistryRejectsDuplicateLabel IMPLEMENTS I_Test
VAR
	Registry	  : TestRegistry<4>;
	First		  : FakeTest;
	Second		  : FakeTest;
	Budgets		  : ST_TestBudgets;
	ExpectedFault : E_RegistrationFault;
	ActualFault	  : E_RegistrationFault;
	ExpectedCount : UDINT;
	ActualCount	  : UDINT;
END_VAR

METHOD Run : BOOL
VAR_INPUT
	Enable : BOOL;
	Test   : I_TestAssertions;
END_VAR
ActualFault	  := Registry.TryClaim(First, 'Homes the axis', Budgets);
ExpectedFault := E_RegistrationFault.None;
Test.AssertEqual(ExpectedFault, ActualFault, 'first accepted');
ActualFault	  := Registry.TryClaim(Second, 'Homes the axis', Budgets);
ExpectedFault := E_RegistrationFault.DuplicateLabel;
Test.AssertEqual(ExpectedFault, ActualFault, 'duplicate refused');
ExpectedCount := 1;
ActualCount	  := Registry.Count;
Test.AssertEqual(ExpectedCount, ActualCount, 'duplicate took no slot');
Run := TRUE;
END_METHOD

END_FUNCTION_BLOCK

// ---- Tests/Registry/TEST_RegistryRejectsEmptyLabelAndNullTest.TcPOU
// Two different mistakes with two different answers. Folding them together would

// send the reader to the wrong argument: an empty label is usually a missing

// string, a null test a missing instance.
FUNCTION_BLOCK TEST_RegistryRejectsEmptyLabelAndNullTest IMPLEMENTS I_Test
VAR
	Registry	  : TestRegistry<4>;
	Fake		  : FakeTest;
	NoTestRef	  : I_Test;
	Budgets		  : ST_TestBudgets;
	ExpectedFault : E_RegistrationFault;
	ActualFault	  : E_RegistrationFault;
	ExpectedCount : UDINT;
	ActualCount	  : UDINT;
END_VAR

METHOD Run : BOOL
VAR_INPUT
	Enable : BOOL;
	Test   : I_TestAssertions;
END_VAR
ActualFault	  := Registry.TryClaim(Fake, '', Budgets);
ExpectedFault := E_RegistrationFault.EmptyLabel;
Test.AssertEqual(ExpectedFault, ActualFault, 'empty label refused');
ActualFault	  := Registry.TryClaim(NoTestRef, 'Has a label but no test', Budgets);
ExpectedFault := E_RegistrationFault.NoTest;
Test.AssertEqual(ExpectedFault, ActualFault, 'null test refused as NoTest');
ExpectedCount := 0;
ActualCount	  := Registry.Count;
Test.AssertEqual(ExpectedCount, ActualCount, 'neither took a slot');
Run := TRUE;
END_METHOD

END_FUNCTION_BLOCK

// ---- Tests/Registry/TEST_RegistryClosesRegistration.TcPOU
// Registration is open until the suite is first enabled, then closed for good. A

// re-run re-executes the registered set; it does not redefine it.

//

// Closed outranks a free slot: refusing a late claim as Full would be a lie.
FUNCTION_BLOCK TEST_RegistryClosesRegistration IMPLEMENTS I_Test
VAR
	Registry	  : TestRegistry<4>;
	Early		  : FakeTest;
	Late		  : FakeTest;
	Budgets		  : ST_TestBudgets;
	ExpectedFault : E_RegistrationFault;
	ActualFault	  : E_RegistrationFault;
	ExpectedCount : UDINT;
	ActualCount	  : UDINT;
END_VAR

METHOD Run : BOOL
VAR_INPUT
	Enable : BOOL;
	Test   : I_TestAssertions;
END_VAR
Test.AssertTrue(Registry.IsOpen, 'open before Close');
ActualFault	  := Registry.TryClaim(Early, 'Registered in time', Budgets);
ExpectedFault := E_RegistrationFault.None;
Test.AssertEqual(ExpectedFault, ActualFault, 'accepted while open');
Registry.Close();
Test.AssertFalse(Registry.IsOpen, 'closed after Close');
ActualFault	  := Registry.TryClaim(Late, 'Registered too late', Budgets);
ExpectedFault := E_RegistrationFault.Closed;
Test.AssertEqual(ExpectedFault, ActualFault, 'refused as Closed, not Full');
ExpectedCount := 1;
ActualCount	  := Registry.Count;
Test.AssertEqual(ExpectedCount, ActualCount, 'late claim took no slot');
Run := TRUE;
END_METHOD

END_FUNCTION_BLOCK

// ---- Tests/Registry/TEST_RegistryLookup.TcPOU
// Lookup answers with an index or -1. ReRunSingle depends on both answers.

//

// An empty label must not match an unclaimed slot, whose label is also empty.
FUNCTION_BLOCK TEST_RegistryLookup IMPLEMENTS I_Test
VAR
	Registry	  : TestRegistry<4>;
	Fakes		  : ARRAY[0..2] OF FakeTest;
	Budgets		  : ST_TestBudgets;
	ExpectedIndex : DINT;
	ActualIndex	  : DINT;
END_VAR

METHOD Run : BOOL
VAR_INPUT
	Enable : BOOL;
	Test   : I_TestAssertions;
END_VAR
Registry.TryClaim(Fakes[0], 'Alpha', Budgets);
Registry.TryClaim(Fakes[1], 'Beta', Budgets);
Registry.TryClaim(Fakes[2], 'Gamma', Budgets);
ExpectedIndex := 0;
ActualIndex	  := Registry.Lookup('Alpha');
Test.AssertEqual(ExpectedIndex, ActualIndex, 'first label');
ExpectedIndex := 2;
ActualIndex	  := Registry.Lookup('Gamma');
Test.AssertEqual(ExpectedIndex, ActualIndex, 'last label');
ExpectedIndex := -1;
ActualIndex	  := Registry.Lookup('Never registered');
Test.AssertEqual(ExpectedIndex, ActualIndex, 'unknown label is -1');
ExpectedIndex := -1;
ActualIndex	  := Registry.Lookup('');
Test.AssertEqual(ExpectedIndex, ActualIndex, 'empty label is -1');
Run := TRUE;
END_METHOD

END_FUNCTION_BLOCK

// ---- Tests/Registry/TEST_RegistryPreservesOrder.TcPOU
// Order of registration is order of execution. Nothing sorts, and a refusal in

// the middle must not reorder what came before or after it.
FUNCTION_BLOCK TEST_RegistryPreservesOrder IMPLEMENTS I_Test
VAR
	Registry	  : TestRegistry<4>;
	Fakes		  : ARRAY[0..2] OF FakeTest;
	Rejected	  : FakeTest;
	Budgets		  : ST_TestBudgets;
	Slot		  : ST_TestSlot;
	ExpectedLabel : T_MaxString;
	ActualLabel	  : T_MaxString;
END_VAR

METHOD Run : BOOL
VAR_INPUT
	Enable : BOOL;
	Test   : I_TestAssertions;
END_VAR
Registry.TryClaim(Fakes[0], 'Zulu', Budgets);
Registry.TryClaim(Rejected, 'Zulu', Budgets);
Registry.TryClaim(Fakes[1], 'Yankee', Budgets);
Registry.TryClaim(Fakes[2], 'Xray', Budgets);
Slot		  := Registry.Slot(0);
ActualLabel	  := Slot.Label;
ExpectedLabel := 'Zulu';
Test.AssertEqual(ExpectedLabel, ActualLabel, 'slot 0');
Slot		  := Registry.Slot(1);
ActualLabel	  := Slot.Label;
ExpectedLabel := 'Yankee';
Test.AssertEqual(ExpectedLabel, ActualLabel, 'slot 1 unaffected by the refusal');
Slot		  := Registry.Slot(2);
ActualLabel	  := Slot.Label;
ExpectedLabel := 'Xray';
Test.AssertEqual(ExpectedLabel, ActualLabel, 'slot 2');
Slot		  := Registry.Slot(3);
ActualLabel	  := Slot.Label;
ExpectedLabel := '';
Test.AssertEqual(ExpectedLabel, ActualLabel, 'unclaimed index is an empty slot');
Run := TRUE;
END_METHOD

END_FUNCTION_BLOCK

// ---- Tests/Registry/TEST_RegistrySlotCarriesItsIndex.TcPOU
// A slot knows where it lives, so a holder of the slot reaches the matching

// journal without carrying a second value alongside it. An unclaimed slot reports

// -1, the same "nothing here" answer its null Test gives.
FUNCTION_BLOCK TEST_RegistrySlotCarriesItsIndex IMPLEMENTS I_Test
VAR
	Registry	  : TestRegistry<3>;
	Fakes		  : ARRAY[0..1] OF FakeTest;
	Budgets		  : ST_TestBudgets;
	Slot		  : ST_TestSlot;
	ExpectedIndex : DINT;
	ActualIndex	  : DINT;
END_VAR

METHOD Run : BOOL
VAR_INPUT
	Enable : BOOL;
	Test   : I_TestAssertions;
END_VAR
Registry.TryClaim(Fakes[0], 'First', Budgets);
Registry.TryClaim(Fakes[1], 'Second', Budgets);
Slot		  := Registry.Slot(0);
ExpectedIndex := 0;
ActualIndex	  := Slot.Index;
Test.AssertEqual(ExpectedIndex, ActualIndex, 'slot 0 knows it is 0');
Slot		  := Registry.Slot(1);
ExpectedIndex := 1;
ActualIndex	  := Slot.Index;
Test.AssertEqual(ExpectedIndex, ActualIndex, 'slot 1 knows it is 1');
Slot		  := Registry.Slot(2);
ExpectedIndex := -1;
ActualIndex	  := Slot.Index;
Test.AssertEqual(ExpectedIndex, ActualIndex, 'unclaimed slot is -1');
Test.AssertTrue(Slot.Test = 0, 'and carries no test');
Run := TRUE;
END_METHOD

END_FUNCTION_BLOCK

// ---- Tests/Registry/TEST_RegistryResolvesOptionalHooks.TcPOU
// The three optional hooks are resolved once, at registration, and

// independently. A test implementing one must not appear to implement the others.
FUNCTION_BLOCK TEST_RegistryResolvesOptionalHooks IMPLEMENTS I_Test
VAR
	Registry  : TestRegistry<4>;
	Bare	  : FakeTest;
	SetupOnly : FakeTestWithSetup;
	AllHooks  : FakeTestWithAllHooks;
	Budgets	  : ST_TestBudgets;
	Slot	  : ST_TestSlot;
END_VAR

METHOD Run : BOOL
VAR_INPUT
	Enable : BOOL;
	Test   : I_TestAssertions;
END_VAR
Registry.TryClaim(Bare, 'Implements nothing optional', Budgets);
Registry.TryClaim(SetupOnly, 'Implements setup only', Budgets);
Registry.TryClaim(AllHooks, 'Implements everything', Budgets);
Slot := Registry.Slot(0);
Test.AssertTrue(Slot.Setup = 0, 'bare: no setup');
Test.AssertTrue(Slot.Teardown = 0, 'bare: no teardown');
Test.AssertTrue(Slot.Location = 0, 'bare: no location');
Slot := Registry.Slot(1);
Test.AssertTrue(Slot.Setup <> 0, 'setup only: setup resolved');
Test.AssertTrue(Slot.Teardown = 0, 'setup only: teardown still null');
Test.AssertTrue(Slot.Location = 0, 'setup only: location still null');
Slot := Registry.Slot(2);
Test.AssertTrue(Slot.Setup <> 0, 'all hooks: setup');
Test.AssertTrue(Slot.Teardown <> 0, 'all hooks: teardown');
Test.AssertTrue(Slot.Location <> 0, 'all hooks: location');
Run := TRUE;
END_METHOD

END_FUNCTION_BLOCK

// ---- Doubles/FakeTestWithSetup.TcPOU
// Implements ONE optional hook and not the other two.

//

// The case that matters for hook resolution: the three are independent, so

// resolving one must not resolve the others. A registry that queried once and

// reused the answer would pass with FakeTest and with FakeTestWithAllHooks, and

// fail only here.
FUNCTION_BLOCK FakeTestWithSetup IMPLEMENTS I_Test, I_TestSetup
VAR
	_RunCount : UDINT;
END_VAR

METHOD Run : BOOL
VAR_INPUT
	Enable : BOOL;
	Test   : I_TestAssertions;
END_VAR
_RunCount := _RunCount + 1;
Run		  := TRUE;
END_METHOD

METHOD Setup : BOOL
VAR_INPUT
	Enable : BOOL;
	Test   : I_TestAssertions;
END_VAR
Setup := TRUE;
END_METHOD

END_FUNCTION_BLOCK

// ---- Doubles/FakeTestWithAllHooks.TcPOU
// Implements every optional hook, so all three must resolve non-null.
FUNCTION_BLOCK FakeTestWithAllHooks IMPLEMENTS I_Test, I_TestSetup, I_TestTeardown, I_TestLocation
VAR
	_RunCount : UDINT;
END_VAR

PROPERTY Path : T_MaxString
GET
Path := 'Verifier.Doubles.AllHooks';
END_GET
END_PROPERTY

METHOD Run : BOOL
VAR_INPUT
	Enable : BOOL;
	Test   : I_TestAssertions;
END_VAR
_RunCount := _RunCount + 1;
Run		  := TRUE;
END_METHOD

METHOD Setup : BOOL
VAR_INPUT
	Enable : BOOL;
	Test   : I_TestAssertions;
END_VAR
Setup := TRUE;
END_METHOD

METHOD Teardown : BOOL
VAR_INPUT
	Enable : BOOL;
	Test   : I_TestAssertions;
END_VAR
Teardown := TRUE;
END_METHOD

END_FUNCTION_BLOCK

// ---- Tests/Registry/TEST_RegistryJournalsArePerSlot.TcPOU
// Every registered test gets its own journal, and Journal() hands back a LIVE

// reference rather than a copy - a copy would record into something nobody reads.
FUNCTION_BLOCK TEST_RegistryJournalsArePerSlot IMPLEMENTS I_Test
VAR
	Registry	  : TestRegistry<4>;
	Fakes		  : ARRAY[0..1] OF FakeTest;
	Budgets		  : ST_TestBudgets;
	JournalA	  : REFERENCE TO TestJournal;
	JournalB	  : REFERENCE TO TestJournal;
	ExpectedLabel : T_MaxString;
	ActualLabel	  : T_MaxString;
END_VAR

METHOD Run : BOOL
VAR_INPUT
	Enable : BOOL;
	Test   : I_TestAssertions;
END_VAR
Registry.TryClaim(Fakes[0], 'First', Budgets);
Registry.TryClaim(Fakes[1], 'Second', Budgets);
JournalA REF= Registry.Journal(0);
JournalB REF= Registry.Journal(1);
Test.AssertTrue(__ISVALIDREF(JournalA), 'journal 0 is valid');
Test.AssertTrue(__ISVALIDREF(JournalB), 'journal 1 is valid');

// Written through the returned reference. If it were a copy, nothing below would

// read back what was written here.
JournalA.Begin('First', 'Verifier.First');
JournalB.Begin('Second', 'Verifier.Second');

// Re-fetched, not reused: reading back through a FRESH reference proves the

// write reached the registry's storage rather than a local alias.

//

// A member cannot be read off a call result in TwinCAT, so each reference is

// taken into a variable first.
JournalA	  REF= Registry.Journal(0);
ActualLabel	  := JournalA.Label;
ExpectedLabel := 'First';
Test.AssertEqual(ExpectedLabel, ActualLabel, 'journal 0 kept its write');
JournalB	  REF= Registry.Journal(1);
ActualLabel	  := JournalB.Label;
ExpectedLabel := 'Second';
Test.AssertEqual(ExpectedLabel, ActualLabel, 'journal 1 is a different object');
Run := TRUE;
END_METHOD

END_FUNCTION_BLOCK

// ---- Tests/Registry/TEST_RegistryJournalRejectsBadIndex.TcPOU
// An index outside the registered range yields an INVALID reference, not a live

// one pointing at whatever was nearby.

//

// A method returning REFERENCE TO that simply returns leaves the reference

// undefined, and undefined reads as valid often enough to pass by luck. Journal

// assigns REF= 0 first, and this is what holds that in place.
FUNCTION_BLOCK TEST_RegistryJournalRejectsBadIndex IMPLEMENTS I_Test
VAR
	Registry : TestRegistry<4>;
	Fake	 : FakeTest;
	Budgets	 : ST_TestBudgets;
	Borrowed : REFERENCE TO TestJournal;
END_VAR

METHOD Run : BOOL
VAR_INPUT
	Enable : BOOL;
	Test   : I_TestAssertions;
END_VAR
Registry.TryClaim(Fake, 'The only one', Budgets);
Borrowed REF= Registry.Journal(0);
Test.AssertTrue(__ISVALIDREF(Borrowed), 'registered index is valid');
Borrowed REF= Registry.Journal(1);
Test.AssertFalse(__ISVALIDREF(Borrowed), 'unclaimed index is invalid');
Borrowed REF= Registry.Journal(-1);
Test.AssertFalse(__ISVALIDREF(Borrowed), 'negative index is invalid');
Run := TRUE;
END_METHOD

END_FUNCTION_BLOCK

// ---- Tests/Arbiter/TEST_ArbiterVisitsEveryTestOnce.TcPOU
// Registration order is execution order, every test is visited exactly once, and

// the pass ends by saying so rather than by wrapping round.
FUNCTION_BLOCK TEST_ArbiterVisitsEveryTestOnce IMPLEMENTS I_Test
VAR
	Registry	  : TestRegistry<3>;
	Arbiter		  : TestArbiter;
	Fakes		  : ARRAY[0..2] OF FakeTest;
	Budgets		  : ST_TestBudgets;
	i			  : DINT;
	Active		  : ST_TestSlot;
	ExpectedIndex : DINT;
	ActualIndex	  : DINT;
	ExpectedLabel : T_MaxString;
	ActualLabel	  : T_MaxString;
END_VAR

METHOD Run : BOOL
VAR_INPUT
	Enable : BOOL;
	Test   : I_TestAssertions;
END_VAR
Registry.TryClaim(Fakes[0], 'Alpha', Budgets);
Registry.TryClaim(Fakes[1], 'Beta', Budgets);
Registry.TryClaim(Fakes[2], 'Gamma', Budgets);
Arbiter.Attach(Registry);
Arbiter.Begin();
FOR i := 0 TO 2 DO
	Test.AssertTrue(Arbiter.Advance(), 'advance to a test');
	Test.AssertTrue(Arbiter.HasCurrent, 'a test is active');
	Active		  := Arbiter.Current;
	ExpectedIndex := i;
	ActualIndex	  := Active.Index;
	Test.AssertEqual(ExpectedIndex, ActualIndex, 'slot carries its index');
END_FOR

ActualLabel	  := Active.Label;
ExpectedLabel := 'Gamma';
Test.AssertEqual(ExpectedLabel, ActualLabel, 'visited in registration order');
Test.AssertFalse(Arbiter.Advance(), 'no fourth test');
Test.AssertTrue(Arbiter.IsExhausted, 'exhausted');
Test.AssertFalse(Arbiter.Advance(), 'and stays exhausted');
Run := TRUE;
END_METHOD

END_FUNCTION_BLOCK

// ---- Tests/Arbiter/TEST_ArbiterCurrentIsNullWhenNothingActive.TcPOU
// "Nothing active" is a NULL REFERENCE, not a sentinel index. The original let

// index 0 double as "none", so a caller reading the index without asking first

// got a live test that was not running.
FUNCTION_BLOCK TEST_ArbiterCurrentIsNullWhenNothingActive IMPLEMENTS I_Test
VAR
	Registry	  : TestRegistry<3>;
	Arbiter		  : TestArbiter;
	Fakes		  : ARRAY[0..2] OF FakeTest;
	Budgets		  : ST_TestBudgets;
	Active		  : ST_TestSlot;
	ExpectedIndex : DINT;
	ActualIndex	  : DINT;
END_VAR

METHOD Run : BOOL
VAR_INPUT
	Enable : BOOL;
	Test   : I_TestAssertions;
END_VAR
Registry.TryClaim(Fakes[0], 'Alpha', Budgets);
Registry.TryClaim(Fakes[1], 'Beta', Budgets);
Arbiter.Attach(Registry);
Arbiter.Begin();
Active := Arbiter.Current;
Test.AssertTrue(Active.Test = 0, 'no test after Begin');
Test.AssertFalse(Arbiter.HasCurrent, 'HasCurrent agrees');
ExpectedIndex := -1;
ActualIndex	  := Active.Index;
Test.AssertEqual(ExpectedIndex, ActualIndex, 'index is -1, not 0');
Arbiter.Advance();
Active := Arbiter.Current;
Test.AssertTrue(Active.Test <> 0, 'a real test once advanced');
Run := TRUE;
END_METHOD

END_FUNCTION_BLOCK

// ---- Tests/Arbiter/TEST_ArbiterEmptyPassIsComplete.TcPOU
// A suite with nothing registered is COMPLETE, not stuck. If it reported

// otherwise, any sequencer aggregating it would wait for it forever.

//

// An arbiter never attached at all is also an empty pass, not a fault: a suite

// that was never wired up should complete rather than hang what is above it.
FUNCTION_BLOCK TEST_ArbiterEmptyPassIsComplete IMPLEMENTS I_Test
VAR
	Registry   : TestRegistry<3>;
	Arbiter	   : TestArbiter;
	Unattached : TestArbiter;
END_VAR

METHOD Run : BOOL
VAR_INPUT
	Enable : BOOL;
	Test   : I_TestAssertions;
END_VAR
Arbiter.Attach(Registry);
Arbiter.Begin();
Test.AssertTrue(Arbiter.IsExhausted, 'exhausted immediately');
Test.AssertFalse(Arbiter.HasCurrent, 'nothing active');
Test.AssertFalse(Arbiter.Advance(), 'nothing to advance to');
Test.AssertTrue(Arbiter.IsExhausted, 'still exhausted');
Unattached.Begin();
Test.AssertTrue(Unattached.IsExhausted, 'unattached is exhausted');
Test.AssertFalse(Unattached.Advance(), 'unattached advances to nothing');
Run := TRUE;
END_METHOD

END_FUNCTION_BLOCK

// ---- Tests/Arbiter/TEST_ArbiterAbandonEndsThePass.TcPOU
// Dropping Enable abandons the run. The tests not yet reached are NOT visited: a

// run that stopped half way has not been run, and reporting the remainder as

// passed, failed or skipped would be inventing a result.
FUNCTION_BLOCK TEST_ArbiterAbandonEndsThePass IMPLEMENTS I_Test
VAR
	Registry	  : TestRegistry<3>;
	Arbiter		  : TestArbiter;
	Fakes		  : ARRAY[0..2] OF FakeTest;
	Budgets		  : ST_TestBudgets;
	Active		  : ST_TestSlot;
	ExpectedLabel : T_MaxString;
	ActualLabel	  : T_MaxString;
END_VAR

METHOD Run : BOOL
VAR_INPUT
	Enable : BOOL;
	Test   : I_TestAssertions;
END_VAR
Registry.TryClaim(Fakes[0], 'Alpha', Budgets);
Registry.TryClaim(Fakes[1], 'Beta', Budgets);
Registry.TryClaim(Fakes[2], 'Gamma', Budgets);
Arbiter.Attach(Registry);
Arbiter.Begin();
Arbiter.Advance();
Active		  := Arbiter.Current;
ActualLabel	  := Active.Label;
ExpectedLabel := 'Alpha';
Test.AssertEqual(ExpectedLabel, ActualLabel, 'first test active');
Arbiter.Abandon();
Test.AssertFalse(Arbiter.HasCurrent, 'nothing active after Abandon');
Test.AssertTrue(Arbiter.IsExhausted, 'pass is over');
Test.AssertFalse(Arbiter.Advance(), 'Beta and Gamma are not visited');
Run := TRUE;
END_METHOD

END_FUNCTION_BLOCK

// ---- Tests/Arbiter/TEST_ArbiterNotExhaustedWhileLastTestRuns.TcPOU
// IsExhausted needs BOTH conditions: nothing left to hand out AND nothing

// running. After the last test is selected there is nothing left to give, but that

// test is still going - reporting the suite complete there would cut it off

// mid-run and lose its verdict.
FUNCTION_BLOCK TEST_ArbiterNotExhaustedWhileLastTestRuns IMPLEMENTS I_Test
VAR
	Registry : TestRegistry<3>;
	Arbiter	 : TestArbiter;
	Fakes	 : ARRAY[0..2] OF FakeTest;
	Budgets	 : ST_TestBudgets;
END_VAR

METHOD Run : BOOL
VAR_INPUT
	Enable : BOOL;
	Test   : I_TestAssertions;
END_VAR
Registry.TryClaim(Fakes[0], 'Only one', Budgets);
Arbiter.Attach(Registry);
Arbiter.Begin();
Arbiter.Advance();
Test.AssertTrue(Arbiter.HasCurrent, 'the one test is running');
Test.AssertFalse(Arbiter.IsExhausted, 'NOT exhausted while it runs');
Arbiter.Advance();
Test.AssertFalse(Arbiter.HasCurrent, 'nothing running now');
Test.AssertTrue(Arbiter.IsExhausted, 'exhausted once it is done');
Run := TRUE;
END_METHOD

END_FUNCTION_BLOCK

// ---- Tests/Arbiter/TEST_ArbiterRestartsFromTheBeginning.TcPOU
// Begin is also what a re-run calls. A re-run re-executes the registered set from

// the start, so there is no separate restart path that could drift out of step

// with this one.
FUNCTION_BLOCK TEST_ArbiterRestartsFromTheBeginning IMPLEMENTS I_Test
VAR
	Registry	  : TestRegistry<3>;
	Arbiter		  : TestArbiter;
	Fakes		  : ARRAY[0..2] OF FakeTest;
	Budgets		  : ST_TestBudgets;
	Active		  : ST_TestSlot;
	ExpectedLabel : T_MaxString;
	ActualLabel	  : T_MaxString;
END_VAR

METHOD Run : BOOL
VAR_INPUT
	Enable : BOOL;
	Test   : I_TestAssertions;
END_VAR
Registry.TryClaim(Fakes[0], 'Alpha', Budgets);
Registry.TryClaim(Fakes[1], 'Beta', Budgets);
Arbiter.Attach(Registry);
Arbiter.Begin();
Arbiter.Advance();
Arbiter.Advance();
Arbiter.Advance();
Test.AssertTrue(Arbiter.IsExhausted, 'first pass finished');
Arbiter.Begin();
Test.AssertFalse(Arbiter.IsExhausted, 'exhausted state cleared');
Test.AssertTrue(Arbiter.Advance(), 'advances again');
Active		  := Arbiter.Current;
ActualLabel	  := Active.Label;
ExpectedLabel := 'Alpha';
Test.AssertEqual(ExpectedLabel, ActualLabel, 'back at the first test');
Run := TRUE;
END_METHOD

END_FUNCTION_BLOCK

// ---- Tests/Verdict/TEST_VerdictRecordsAFailure.TcPOU
// The failure path, exercised deliberately.

//

// Sixteen green tests prove nothing if a check cannot go red. This drives a

// mismatched AssertEqual into a private journal and asserts the journal noticed.
FUNCTION_BLOCK TEST_VerdictRecordsAFailure IMPLEMENTS I_Test
VAR
	// A private journal and handle, so a DELIBERATE failure can be recorded and

	// inspected without the suite's own verdict ever seeing it. The test itself

	// passes; what it proves is that failing works.
	Subject		   : TestJournal;
	Handle		   : TestVerdict;
	ExpectedValue  : DINT := 1;
	ActualValue	   : DINT := 2;
	ExpectedKind   : E_FailureKind;
	ActualKind	   : E_FailureKind;
	ExpectedStatus : E_TestStatus;
	ActualStatus   : E_TestStatus;
	ExpectedCount  : UDINT;
	ActualCount	   : UDINT;
END_VAR

METHOD Run : BOOL
VAR_INPUT
	Enable : BOOL;
	Test   : I_TestAssertions;
END_VAR
Handle.Target(Subject);
Subject.Begin('deliberate', '');

// 1 <> 2. If this records a pass, every result in this project is worthless.
Handle.AssertEqual(ExpectedValue, ActualValue, 'one is not two');
ExpectedCount := 1;
ActualCount	  := Subject.AssertionCount;
Test.AssertEqual(ExpectedCount, ActualCount, 'the check was counted');
ExpectedKind := E_FailureKind.ValueMismatch;
ActualKind	 := Subject.Kind;
Test.AssertEqual(ExpectedKind, ActualKind, 'recorded as a value mismatch');

// Passed is what the runner asks for when a body returns TRUE. A recorded failure

// must override it.
Subject.Finish(E_TestStatus.Passed);
ExpectedStatus := E_TestStatus.Failed;
ActualStatus   := Subject.Status;
Test.AssertEqual(ExpectedStatus, ActualStatus, 'a recorded failure overrides Passed');
Handle.Untarget();
Run := TRUE;
END_METHOD

END_FUNCTION_BLOCK

// ---- Tests/Verdict/TEST_VerdictPassDoesNotOvertakeAFailure.TcPOU
// The verdict cannot return to Passed once a check has failed. Later checks are

// still evaluated and counted - a run should report everything it found, not stop

// at the first problem - but none of them can undo the first failure.
FUNCTION_BLOCK TEST_VerdictPassDoesNotOvertakeAFailure IMPLEMENTS I_Test
VAR
	// A private journal and handle, so a DELIBERATE failure can be recorded and

	// inspected without the suite's own verdict ever seeing it. The test itself

	// passes; what it proves is that failing works.
	Subject		   : TestJournal;
	Handle		   : TestVerdict;
	Same		   : DINT := 7;
	Lower		   : DINT := 1;
	Higher		   : DINT := 2;
	ExpectedStatus : E_TestStatus;
	ActualStatus   : E_TestStatus;
	ExpectedCount  : UDINT;
	ActualCount	   : UDINT;
END_VAR

METHOD Run : BOOL
VAR_INPUT
	Enable : BOOL;
	Test   : I_TestAssertions;
END_VAR
Handle.Target(Subject);
Subject.Begin('deliberate', '');
Handle.AssertEqual(Lower, Higher, 'fails first');
Handle.AssertEqual(Same, Same, 'passes second');
Handle.AssertTrue(TRUE, 'passes third');
ExpectedCount := 3;
ActualCount	  := Subject.AssertionCount;
Test.AssertEqual(ExpectedCount, ActualCount, 'every check was evaluated');
Subject.Finish(E_TestStatus.Passed);
ExpectedStatus := E_TestStatus.Failed;
ActualStatus   := Subject.Status;
Test.AssertEqual(ExpectedStatus, ActualStatus, 'still Failed after two passes');
Handle.Untarget();
Run := TRUE;
END_METHOD

END_FUNCTION_BLOCK

// ---- Tests/Verdict/TEST_VerdictZeroChecksIsErrored.TcPOU
// A test that finishes having recorded NOTHING is Errored, not Passed.

//

// A body that checked nothing usually means a branch never ran. Reporting that

// green is a silent false pass wearing a badge, and it is one of the defects this

// library was rewritten to remove.
FUNCTION_BLOCK TEST_VerdictZeroChecksIsErrored IMPLEMENTS I_Test
VAR
	// A private journal and handle, so a DELIBERATE failure can be recorded and

	// inspected without the suite's own verdict ever seeing it. The test itself

	// passes; what it proves is that failing works.
	Subject		   : TestJournal;
	Handle		   : TestVerdict;
	ExpectedStatus : E_TestStatus;
	ActualStatus   : E_TestStatus;
END_VAR

METHOD Run : BOOL
VAR_INPUT
	Enable : BOOL;
	Test   : I_TestAssertions;
END_VAR
Handle.Target(Subject);
Subject.Begin('checked nothing', '');

// No checks at all, then the runner asks for Passed.
Subject.Finish(E_TestStatus.Passed);
ExpectedStatus := E_TestStatus.Errored;
ActualStatus   := Subject.Status;
Test.AssertEqual(ExpectedStatus, ActualStatus, 'no checks means Errored, not Passed');
Handle.Untarget();
Run := TRUE;
END_METHOD

END_FUNCTION_BLOCK

// ---- Tests/Verdict/TEST_VerdictReportErrorIsNotAFailure.TcPOU
// Errored is distinct from Failed: the code under test was never shown to be

// wrong. A precondition was absent or a target unreachable.

//

// Conflating them sends whoever reads the report hunting a defect that is not

// there.
FUNCTION_BLOCK TEST_VerdictReportErrorIsNotAFailure IMPLEMENTS I_Test
VAR
	// A private journal and handle, so a DELIBERATE failure can be recorded and

	// inspected without the suite's own verdict ever seeing it. The test itself

	// passes; what it proves is that failing works.
	Subject		   : TestJournal;
	Handle		   : TestVerdict;
	ExpectedStatus : E_TestStatus;
	ActualStatus   : E_TestStatus;
	ExpectedKind   : E_FailureKind;
	ActualKind	   : E_FailureKind;
END_VAR

METHOD Run : BOOL
VAR_INPUT
	Enable : BOOL;
	Test   : I_TestAssertions;
END_VAR
Handle.Target(Subject);
Subject.Begin('could not run', '');
Handle.ReportError('the axis would not power');
ExpectedKind := E_FailureKind.Environment;
ActualKind	 := Subject.Kind;
Test.AssertEqual(ExpectedKind, ActualKind, 'recorded as environmental');
Subject.Finish(E_TestStatus.Passed);
ExpectedStatus := E_TestStatus.Errored;
ActualStatus   := Subject.Status;
Test.AssertEqual(ExpectedStatus, ActualStatus, 'Errored, not Failed');
Handle.Untarget();
Run := TRUE;
END_METHOD

END_FUNCTION_BLOCK

// ---- Tests/Verdict/TEST_VerdictFailIsAPlainFailure.TcPOU
// Fail is the outright failure with no comparison behind it - for a branch that

// should have been unreachable. It is a Failed verdict, not an Errored one:

// reaching that branch IS the code being wrong.
FUNCTION_BLOCK TEST_VerdictFailIsAPlainFailure IMPLEMENTS I_Test
VAR
	// A private journal and handle, so a DELIBERATE failure can be recorded and

	// inspected without the suite's own verdict ever seeing it. The test itself

	// passes; what it proves is that failing works.
	Subject		   : TestJournal;
	Handle		   : TestVerdict;
	ExpectedStatus : E_TestStatus;
	ActualStatus   : E_TestStatus;
END_VAR

METHOD Run : BOOL
VAR_INPUT
	Enable : BOOL;
	Test   : I_TestAssertions;
END_VAR
Handle.Target(Subject);
Subject.Begin('unreachable branch', '');
Handle.Fail('the default case was reached');
Subject.Finish(E_TestStatus.Passed);
ExpectedStatus := E_TestStatus.Failed;
ActualStatus   := Subject.Status;
Test.AssertEqual(ExpectedStatus, ActualStatus, 'Fail produces Failed');
Handle.Untarget();
Run := TRUE;
END_METHOD

END_FUNCTION_BLOCK

// ---- Tests/Verdict/TEST_VerdictSummaryLeadsWithTheStepLabel.TcPOU
// Timeout is the dominant failure mode for anything multi-scan, and there the

// step label IS the diagnostic. "Home: timed out after 5000 cycles" usually ends

// an investigation; "timed out after 5000 cycles" starts one.

//

// The step captured is the one current when the check ran, so a later step cannot

// relabel an earlier failure.
FUNCTION_BLOCK TEST_VerdictSummaryLeadsWithTheStepLabel IMPLEMENTS I_Test
VAR
	// A private journal and handle, so a DELIBERATE failure can be recorded and

	// inspected without the suite's own verdict ever seeing it. The test itself

	// passes; what it proves is that failing works.
	Subject : TestJournal;
	Handle	: TestVerdict;
	Lower	: DINT := 1;
	Higher	: DINT := 2;
	Summary : T_MaxString;
	FoundAt : INT;
END_VAR

METHOD Run : BOOL
VAR_INPUT
	Enable : BOOL;
	Test   : I_TestAssertions;
END_VAR
Handle.Target(Subject);
Subject.Begin('stepped', '');
Handle.SetStep('Home');
Handle.AssertEqual(Lower, Higher, 'while homing');

// A later step must not relabel the failure already recorded.
Handle.SetStep('Retract');
Subject.Finish(E_TestStatus.Passed);
Summary := Subject.Summary;
FoundAt := FIND(Summary, 'Home');
Test.AssertTrue(FoundAt = 1, 'summary opens with the step that was current');
FoundAt := FIND(Summary, 'Retract');
Test.AssertTrue(FoundAt = 0, 'the later step did not relabel it');
Handle.Untarget();
Run := TRUE;
END_METHOD

END_FUNCTION_BLOCK

// ---- Tests/Verdict/TEST_VerdictFirstFailureWinsTheSummary.TcPOU
// Only the FIRST failure's text reaches the 80-character summary. A later failure

// is usually downstream of the first, and the summary has room for one - the rest

// survive on the detail sink.
FUNCTION_BLOCK TEST_VerdictFirstFailureWinsTheSummary IMPLEMENTS I_Test
VAR
	// A private journal and handle, so a DELIBERATE failure can be recorded and

	// inspected without the suite's own verdict ever seeing it. The test itself

	// passes; what it proves is that failing works.
	Subject : TestJournal;
	Handle	: TestVerdict;
	Lower	: DINT := 1;
	Higher	: DINT := 2;
	Summary : T_MaxString;
END_VAR

METHOD Run : BOOL
VAR_INPUT
	Enable : BOOL;
	Test   : I_TestAssertions;
END_VAR
Handle.Target(Subject);
Subject.Begin('two failures', '');
Handle.AssertEqual(Lower, Higher, 'the first thing that broke');
Handle.Fail('a consequence of the first');
Subject.Finish(E_TestStatus.Passed);
Summary := Subject.Summary;
Test.AssertTrue(FIND(Summary, 'the first thing that broke') > 0, 'first failure is in the summary');
Test.AssertTrue(FIND(Summary, 'a consequence of the first') = 0, 'the second is not');
Handle.Untarget();
Run := TRUE;
END_METHOD

END_FUNCTION_BLOCK

// ---- Tests/Verdict/TEST_VerdictUntargetedHandleIsInert.TcPOU
// A handle pointing at nothing records nothing, rather than writing into whatever

// journal happens to be nearby.

//

// The runner untargets after every test. Without this holding, a stray call from a

// test that kept the handle would land in the NEXT test's record.
FUNCTION_BLOCK TEST_VerdictUntargetedHandleIsInert IMPLEMENTS I_Test
VAR
	// A private journal and handle, so a DELIBERATE failure can be recorded and

	// inspected without the suite's own verdict ever seeing it. The test itself

	// passes; what it proves is that failing works.
	Subject		  : TestJournal;
	Handle		  : TestVerdict;
	ExpectedCount : UDINT;
	ActualCount	  : UDINT;
END_VAR

METHOD Run : BOOL
VAR_INPUT
	Enable : BOOL;
	Test   : I_TestAssertions;
END_VAR
Handle.Target(Subject);
Subject.Begin('inert', '');
Handle.AssertTrue(TRUE, 'one real check');
Handle.Untarget();

// Everything below must reach nothing at all.
Handle.AssertTrue(FALSE, 'must not be recorded');
Handle.Fail('must not be recorded');
Handle.ReportError('must not be recorded');
ExpectedCount := 1;
ActualCount	  := Subject.AssertionCount;
Test.AssertEqual(ExpectedCount, ActualCount, 'nothing landed after Untarget');
Subject.Finish(E_TestStatus.Passed);
Test.AssertTrue(Subject.Status = E_TestStatus.Passed, 'and the verdict is untouched');
Run := TRUE;
END_METHOD

END_FUNCTION_BLOCK

// ---- Tests/Journal/TEST_JournalTimesOutOnCycles.TcPOU
// A body that never finishes must be stopped by the deadline rather than stalling

// the suite. Tick both detects the expiry and records it - the runner only has to

// notice it happened.

//

// Called AFTER the body has run, so a budget of one allows one execution.
FUNCTION_BLOCK TEST_JournalTimesOutOnCycles IMPLEMENTS I_Test
VAR
	Subject		   : TestJournal;
	Budgets		   : ST_TestBudgets;
	Expired		   : BOOL;
	ExpectedKind   : E_FailureKind;
	ActualKind	   : E_FailureKind;
	ExpectedStatus : E_TestStatus;
	ActualStatus   : E_TestStatus;
END_VAR

METHOD Run : BOOL
VAR_INPUT
	Enable : BOOL;
	Test   : I_TestAssertions;
END_VAR
Budgets.Body.Cycles		 := 2;
Budgets.Body.IsCyclesSet := TRUE;
Subject.SetBudgets(Budgets);
Subject.Begin('slow', '');
Expired := Subject.Tick();
Test.AssertFalse(Expired, 'a budget of two survives one scan');
Expired := Subject.Tick();
Test.AssertTrue(Expired, 'and expires on the second');
ExpectedKind := E_FailureKind.Timeout;
ActualKind	 := Subject.Kind;
Test.AssertEqual(ExpectedKind, ActualKind, 'recorded as a timeout');

// Tick finishes the journal itself; the runner does not have to.
ExpectedStatus := E_TestStatus.Failed;
ActualStatus   := Subject.Status;
Test.AssertEqual(ExpectedStatus, ActualStatus, 'terminal without further help');
Expired := Subject.Tick();
Test.AssertFalse(Expired, 'and does not fire twice');
Run := TRUE;
END_METHOD

END_FUNCTION_BLOCK

// ---- Tests/Journal/TEST_JournalZeroBudgetDisablesTheDeadline.TcPOU
// Zero disables. That is why "not specified" needs its own flag and cannot be

// inferred from the value - a long-running rig test may legitimately want no scan

// budget at all.
FUNCTION_BLOCK TEST_JournalZeroBudgetDisablesTheDeadline IMPLEMENTS I_Test
VAR
	Subject : TestJournal;
	Budgets : ST_TestBudgets;
	i		: DINT;
	Expired : BOOL;
END_VAR

METHOD Run : BOOL
VAR_INPUT
	Enable : BOOL;
	Test   : I_TestAssertions;
END_VAR
Budgets.Body.Cycles		 := 0;
Budgets.Body.IsCyclesSet := TRUE;
Subject.SetBudgets(Budgets);
Subject.Begin('unbounded', '');
FOR i := 1 TO 50 DO
	IF Subject.Tick() THEN
		Expired := TRUE;
	END_IF
END_FOR

Test.AssertFalse(Expired, 'a zero budget never expires');
Test.AssertTrue(Subject.Status = E_TestStatus.Running, 'and the test is still going');
Run := TRUE;
END_METHOD

END_FUNCTION_BLOCK

// ---- Tests/Journal/TEST_JournalDefaultsFillOnlyWhatWasNotClaimed.TcPOU
// Each unit is tracked separately on purpose. A test naming its own wall-clock

// budget still inherits the suite's scan budget, and the reverse. A single

// "overridden" flag would break exactly that case and nothing else would notice.
FUNCTION_BLOCK TEST_JournalDefaultsFillOnlyWhatWasNotClaimed IMPLEMENTS I_Test
VAR
	Subject		   : TestJournal;
	Claimed		   : ST_TestBudgets;
	Defaults	   : ST_TestBudgets;
	Got			   : ST_TestBudgets;
	ExpectedCycles : UDINT;
	ActualCycles   : UDINT;
	ExpectedTime   : TIME;
	ActualTime	   : TIME;
END_VAR

METHOD Run : BOOL
VAR_INPUT
	Enable : BOOL;
	Test   : I_TestAssertions;
END_VAR
// The test claims a scan budget and says nothing about wall clock.
Claimed.Body.Cycles		 := 7;
Claimed.Body.IsCyclesSet := TRUE;
Subject.SetBudgets(Claimed);
Defaults.Body.Cycles	   := 999;
Defaults.Body.IsCyclesSet  := TRUE;
Defaults.Body.Timeout	   := T#5S;
Defaults.Body.IsTimeoutSet := TRUE;
Subject.ApplyDefaults(Defaults);
Got			   := Subject.Budgets;
ExpectedCycles := 7;
ActualCycles   := Got.Body.Cycles;
Test.AssertEqual(ExpectedCycles, ActualCycles, 'the claimed scan budget survived');
ExpectedTime := T#5S;
ActualTime	 := Got.Body.Timeout;
Test.AssertEqual(ExpectedTime, ActualTime, 'the unclaimed wall clock was filled in');
Run := TRUE;
END_METHOD

END_FUNCTION_BLOCK

// ---- Tests/Journal/TEST_JournalResetKeepsWhatWasRegistered.TcPOU
// A re-run re-executes the registered set; it does not redefine it. Reset clears

// the verdict and the counts, and keeps the label, the location and the budgets

// the test claimed at registration.
FUNCTION_BLOCK TEST_JournalResetKeepsWhatWasRegistered IMPLEMENTS I_Test
VAR
	Subject		   : TestJournal;
	Handle		   : TestVerdict;
	Budgets		   : ST_TestBudgets;
	Got			   : ST_TestBudgets;
	ExpectedCycles : UDINT;
	ActualCycles   : UDINT;
	ExpectedCount  : UDINT;
	ActualCount	   : UDINT;
END_VAR

METHOD Run : BOOL
VAR_INPUT
	Enable : BOOL;
	Test   : I_TestAssertions;
END_VAR
Budgets.Body.Cycles		 := 11;
Budgets.Body.IsCyclesSet := TRUE;
Subject.SetBudgets(Budgets);
Handle.Target(Subject);
Subject.Begin('first run', 'Verifier.Somewhere');
Handle.Fail('deliberate');
Subject.Finish(E_TestStatus.Passed);
Handle.Untarget();
Test.AssertTrue(Subject.Status = E_TestStatus.Failed, 'failed on the first run');
Subject.Reset();
Test.AssertTrue(Subject.Status = E_TestStatus.NotStarted, 'verdict cleared');
Test.AssertTrue(Subject.Kind = E_FailureKind.None, 'failure kind cleared');
ExpectedCount := 0;
ActualCount	  := Subject.AssertionCount;
Test.AssertEqual(ExpectedCount, ActualCount, 'checks cleared');
Got			   := Subject.Budgets;
ExpectedCycles := 11;
ActualCycles   := Got.Body.Cycles;
Test.AssertEqual(ExpectedCycles, ActualCycles, 'the claimed budget survived the reset');
Run := TRUE;
END_METHOD

END_FUNCTION_BLOCK

// ---- Tests/Journal/TEST_JournalSkippedIsTerminalAndNotRed.TcPOU
// A skipped test is not a failure and must not turn a build red. It is terminal

// immediately: a skipped suite reports complete, or an aggregate containing one

// waits for it forever.
FUNCTION_BLOCK TEST_JournalSkippedIsTerminalAndNotRed IMPLEMENTS I_Test
VAR
	Subject : TestJournal;
	Expired : BOOL;
END_VAR

METHOD Run : BOOL
VAR_INPUT
	Enable : BOOL;
	Test   : I_TestAssertions;
END_VAR
Subject.MarkSkipped();
Test.AssertTrue(Subject.Status = E_TestStatus.Skipped, 'Skipped');
Test.AssertTrue(Subject.Kind = E_FailureKind.None, 'with no failure kind');

// Terminal means Tick does nothing further.
Expired := Subject.Tick();
Test.AssertFalse(Expired, 'a skipped test has no deadline left to expire');
Test.AssertTrue(Subject.Status = E_TestStatus.Skipped, 'and stays Skipped');
Run := TRUE;
END_METHOD

END_FUNCTION_BLOCK

// ---- Tests/Runner/TEST_RunnerDrivesThePhasesInOrder.TcPOU
// Setup, then body, then teardown - each exactly once, in that order.

//

// Order is the whole contract of the three-phase model and nothing else in the

// library checks it. Teardown also reads the verdict, which must already be

// terminal by the time it runs.
FUNCTION_BLOCK TEST_RunnerDrivesThePhasesInOrder IMPLEMENTS I_Test
VAR
	// A private runner, driven one scan per call. The outer test spans scans by

	// returning FALSE, which is exactly the mechanism being verified one level down.
	Registry	   : TestRegistry<1>;
	Runner		   : TestRunner;
	Handle		   : TestVerdict;
	Budgets		   : ST_TestBudgets;
	Journal		   : REFERENCE TO TestJournal;
	Slot		   : ST_TestSlot;
	Outcome		   : E_PhaseOutcome;
	Loaded		   : BOOL;
	Phase		   : DINT;
	Scans		   : DINT;
	Subject		   : OrderedHooksTest;
	ExpectedCount  : UDINT;
	ActualCount	   : UDINT;
	ExpectedStatus : E_TestStatus;
	ActualStatus   : E_TestStatus;
END_VAR

METHOD Run : BOOL
VAR_INPUT
	Enable : BOOL;
	Test   : I_TestAssertions;
END_VAR
Scans := Scans + 1;
IF Scans > 200 THEN
	Test.Fail('the subject never reached a terminal outcome');
	Run := TRUE;
	RETURN;
END_IF

CASE Phase OF
	0:
		Registry.TryClaim(Subject, 'ordered', Budgets);
		Runner.Attach(Roster := Registry, Verdict := Handle);
		Slot   := Registry.Slot(0);
		Loaded := Runner.Load(Slot);
		Phase  := 1;
		Run	   := FALSE;

	1:
		Outcome := Runner.Advance(Enable := TRUE);
		IF Outcome <> E_PhaseOutcome.Running THEN
			Phase := 2;
		END_IF

		Run := FALSE;

	2:
		Test.AssertTrue(Loaded, 'the runner accepted the test');
		Test.AssertTrue(Outcome = E_PhaseOutcome.Finished, 'finished cleanly');
		ExpectedCount := 1;
		ActualCount	  := Subject.SetupCalls;
		Test.AssertEqual(ExpectedCount, ActualCount, 'setup called once');
		ActualCount := Subject.BodyCalls;
		Test.AssertEqual(ExpectedCount, ActualCount, 'body called once');
		ActualCount := Subject.TeardownCalls;
		Test.AssertEqual(ExpectedCount, ActualCount, 'teardown called once');
		Test.AssertTrue(Subject.BodyAfterSetup, 'body ran after setup');
		Test.AssertTrue(Subject.TeardownAfterBody, 'teardown ran after the body');

		// Terminal before teardown, so cleanup can branch on the outcome.
		ExpectedStatus := E_TestStatus.Passed;
		ActualStatus   := Subject.StatusInTeardown;
		Test.AssertEqual(ExpectedStatus, ActualStatus, 'teardown saw a settled verdict');
		Journal REF= Registry.Journal(0);
		IF __ISVALIDREF(Journal) THEN
			ActualStatus := Journal.Status;
			Test.AssertEqual(ExpectedStatus, ActualStatus, 'and the journal agrees');
		END_IF

		Run := TRUE;
END_CASE
END_METHOD

END_FUNCTION_BLOCK

// ---- Doubles/OrderedHooksTest.TcPOU
// Implements all three phases and records the order they were called in.

//

// Setup before body, body before teardown, each exactly once. Order is the whole

// contract and nothing else in the library checks it.
FUNCTION_BLOCK OrderedHooksTest IMPLEMENTS I_Test, I_TestSetup, I_TestTeardown
VAR
	_SetupCalls	   : UDINT;
	_BodyCalls	   : UDINT;
	_TeardownCalls : UDINT;

	// Captured at each phase, so the ORDER is provable and not just the counts.
	_BodyAfterSetup	   : BOOL;
	_TeardownAfterBody : BOOL;
	_StatusInTeardown  : E_TestStatus;
END_VAR

PROPERTY BodyAfterSetup : BOOL
GET
BodyAfterSetup := _BodyAfterSetup;
END_GET
END_PROPERTY

PROPERTY BodyCalls : UDINT
GET
BodyCalls := _BodyCalls;
END_GET
END_PROPERTY

METHOD Run : BOOL
VAR_INPUT
	Enable : BOOL;
	Test   : I_TestAssertions;
END_VAR
IF NOT Enable THEN
	Run := TRUE;
	RETURN;
END_IF

_BodyCalls		:= _BodyCalls + 1;
_BodyAfterSetup := (_SetupCalls > 0);
Test.AssertTrue(TRUE, 'body ran');
Run := TRUE;
END_METHOD

METHOD Setup : BOOL
VAR_INPUT
	Enable : BOOL;
	Test   : I_TestAssertions;
END_VAR
_SetupCalls := _SetupCalls + 1;
Setup		:= TRUE;
END_METHOD

PROPERTY SetupCalls : UDINT
GET
SetupCalls := _SetupCalls;
END_GET
END_PROPERTY

// The verdict as teardown saw it. Terminal by then, whatever it is.
PROPERTY StatusInTeardown : E_TestStatus
GET
StatusInTeardown := _StatusInTeardown;
END_GET
END_PROPERTY

METHOD Teardown : BOOL
VAR_INPUT
	Enable : BOOL;
	Test   : I_TestAssertions;
END_VAR
_TeardownCalls	   := _TeardownCalls + 1;
_TeardownAfterBody := (_BodyCalls > 0);

// Readable here on purpose: cleanup may differ by outcome.
_StatusInTeardown := Test.Status;
Teardown		  := TRUE;
END_METHOD

PROPERTY TeardownAfterBody : BOOL
GET
TeardownAfterBody := _TeardownAfterBody;
END_GET
END_PROPERTY

PROPERTY TeardownCalls : UDINT
GET
TeardownCalls := _TeardownCalls;
END_GET
END_PROPERTY

END_FUNCTION_BLOCK

// ---- Tests/Runner/TEST_RunnerRunsAMultiScanBody.TcPOU
// A body returning FALSE is called again next scan, and only then. Multi-cycle is

// the normal case here, not an awkward one.

//

// ElapsedCycles counts the body, so a three-scan body reports three.
FUNCTION_BLOCK TEST_RunnerRunsAMultiScanBody IMPLEMENTS I_Test
VAR
	// A private runner, driven one scan per call. The outer test spans scans by

	// returning FALSE, which is exactly the mechanism being verified one level down.
	Registry	  : TestRegistry<1>;
	Runner		  : TestRunner;
	Handle		  : TestVerdict;
	Budgets		  : ST_TestBudgets;
	Journal		  : REFERENCE TO TestJournal;
	Slot		  : ST_TestSlot;
	Outcome		  : E_PhaseOutcome;
	Loaded		  : BOOL;
	Phase		  : DINT;
	Scans		  : DINT;
	Subject		  : SpanningTest;
	RunningCount  : DINT;
	ExpectedCount : UDINT;
	ActualCount	  : UDINT;
END_VAR

METHOD Run : BOOL
VAR_INPUT
	Enable : BOOL;
	Test   : I_TestAssertions;
END_VAR
Scans := Scans + 1;
IF Scans > 200 THEN
	Test.Fail('the subject never reached a terminal outcome');
	Run := TRUE;
	RETURN;
END_IF

CASE Phase OF
	0:
		Subject.SetScans(3);
		Registry.TryClaim(Subject, 'spanning', Budgets);
		Runner.Attach(Roster := Registry, Verdict := Handle);
		Slot   := Registry.Slot(0);
		Loaded := Runner.Load(Slot);
		Phase  := 1;
		Run	   := FALSE;

	1:
		Outcome := Runner.Advance(Enable := TRUE);
		IF Outcome = E_PhaseOutcome.Running THEN
			RunningCount := RunningCount + 1;
		ELSE
			Phase := 2;
		END_IF

		Run := FALSE;

	2:
		Test.AssertTrue(Outcome = E_PhaseOutcome.Finished, 'finished');
		ExpectedCount := 3;
		ActualCount	  := Subject.BodyCalls;
		Test.AssertEqual(ExpectedCount, ActualCount, 'the body was called three times');

		// Two Running answers, then the finishing one.
		Test.AssertTrue(RunningCount = 2, 'and reported Running in between');

		// TWO, not three. The journal is ticked AFTER the body runs, so on the body's

		// Nth call it has consumed N-1 scans. The first call reports 0, which is what

		// makes IsFirstCycle and ElapsedCycles agree with each other.
		ExpectedCount := 2;
		ActualCount	  := Subject.CyclesAtFinish;
		Test.AssertEqual(ExpectedCount, ActualCount, 'ElapsedCycles excludes the call in progress');
		Test.AssertTrue(Subject.FirstCycleAtStart, 'the first call was the first cycle');
		Run := TRUE;
END_CASE
END_METHOD

END_FUNCTION_BLOCK

// ---- Doubles/SpanningTest.TcPOU
// A body that takes several scans, like most real tests.

//

// Returns FALSE until it has been called ScansToTake times, then records one check

// and returns TRUE. Counts its calls so the runner can be held to calling it

// exactly that many times - no more, no fewer.
FUNCTION_BLOCK SpanningTest IMPLEMENTS I_Test
VAR
	_ScansToTake	   : UDINT := 3;
	_BodyCalls		   : UDINT;
	_AbandonCalls	   : UDINT;
	_FirstCycleAtStart : BOOL;
	_CyclesAtFinish	   : UDINT;
	_Seen			   : BOOL;
END_VAR

// Calls received with Enable FALSE. Exactly one after an abandon.
PROPERTY AbandonCalls : UDINT
GET
AbandonCalls := _AbandonCalls;
END_GET
END_PROPERTY

PROPERTY BodyCalls : UDINT
GET
BodyCalls := _BodyCalls;
END_GET
END_PROPERTY

// ElapsedCycles the body saw on its last call. Counts the BODY only, not setup.
PROPERTY CyclesAtFinish : UDINT
GET
CyclesAtFinish := _CyclesAtFinish;
END_GET
END_PROPERTY

// I_TestTiming.IsFirstCycle as the body saw it on its first call. TRUE even when

// setup consumed scans first - the body's first scan is the body's first scan.
PROPERTY FirstCycleAtStart : BOOL
GET
FirstCycleAtStart := _FirstCycleAtStart;
END_GET
END_PROPERTY

METHOD Run : BOOL
VAR_INPUT
	Enable : BOOL;
	Test   : I_TestAssertions;
END_VAR
IF NOT Enable THEN
	_AbandonCalls := _AbandonCalls + 1;
	Run			  := TRUE;
	RETURN;
END_IF

_BodyCalls := _BodyCalls + 1;
IF NOT _Seen THEN
	// Captured on the body's FIRST call, whatever setup did beforehand.
	_Seen			   := TRUE;
	_FirstCycleAtStart := Test.IsFirstCycle;
END_IF

IF _BodyCalls < _ScansToTake THEN
	Run := FALSE;
	RETURN;
END_IF

_CyclesAtFinish := Test.ElapsedCycles;
Test.AssertTrue(TRUE, 'reached the end');
Run := TRUE;
END_METHOD

// How many scans the body should take before finishing.
METHOD SetScans
VAR_INPUT
	Scans : UDINT;
END_VAR
_ScansToTake := Scans;
END_METHOD

END_FUNCTION_BLOCK

// ---- Tests/Runner/TEST_RunnerSetupFailureSkipsTheBody.TcPOU
// A failure recorded during setup ends the test WITHOUT running the body, and

// still runs teardown.

//

// The body is what is under test; a fixture that never came up means it was never

// exercised. Reporting that as a failed check would send the reader after the

// wrong thing.
FUNCTION_BLOCK TEST_RunnerSetupFailureSkipsTheBody IMPLEMENTS I_Test
VAR
	// A private runner, driven one scan per call. The outer test spans scans by

	// returning FALSE, which is exactly the mechanism being verified one level down.
	Registry	   : TestRegistry<1>;
	Runner		   : TestRunner;
	Handle		   : TestVerdict;
	Budgets		   : ST_TestBudgets;
	Journal		   : REFERENCE TO TestJournal;
	Slot		   : ST_TestSlot;
	Outcome		   : E_PhaseOutcome;
	Loaded		   : BOOL;
	Phase		   : DINT;
	Scans		   : DINT;
	Subject		   : SetupFailsTest;
	ExpectedZero   : UDINT;
	ExpectedOne	   : UDINT;
	ActualCount	   : UDINT;
	ExpectedStatus : E_TestStatus;
	ActualStatus   : E_TestStatus;
END_VAR

METHOD Run : BOOL
VAR_INPUT
	Enable : BOOL;
	Test   : I_TestAssertions;
END_VAR
Scans := Scans + 1;
IF Scans > 200 THEN
	Test.Fail('the subject never reached a terminal outcome');
	Run := TRUE;
	RETURN;
END_IF

CASE Phase OF
	0:
		Registry.TryClaim(Subject, 'setup fails', Budgets);
		Runner.Attach(Roster := Registry, Verdict := Handle);
		Slot   := Registry.Slot(0);
		Loaded := Runner.Load(Slot);
		Phase  := 1;
		Run	   := FALSE;

	1:
		Outcome := Runner.Advance(Enable := TRUE);
		IF Outcome <> E_PhaseOutcome.Running THEN
			Phase := 2;
		END_IF

		Run := FALSE;

	2:
		ExpectedZero := 0;
		ActualCount	 := Subject.BodyCalls;
		Test.AssertEqual(ExpectedZero, ActualCount, 'the body was never called');
		ExpectedOne := 1;
		ActualCount := Subject.TeardownCalls;
		Test.AssertEqual(ExpectedOne, ActualCount, 'teardown ran anyway');
		Journal REF= Registry.Journal(0);
		IF __ISVALIDREF(Journal) THEN
			ExpectedStatus := E_TestStatus.Failed;
			ActualStatus   := Journal.Status;
			Test.AssertEqual(ExpectedStatus, ActualStatus, 'the verdict is Failed');
		END_IF

		Run := TRUE;
END_CASE
END_METHOD

END_FUNCTION_BLOCK

// ---- Doubles/SetupFailsTest.TcPOU
// Setup records a failure and completes. The body must NEVER be called - a test

// whose fixture never came up has not been exercised, and reporting it as a failed

// check would be a lie - but teardown must still run.
FUNCTION_BLOCK SetupFailsTest IMPLEMENTS I_Test, I_TestSetup, I_TestTeardown
VAR
	_BodyCalls	   : UDINT;
	_TeardownCalls : UDINT;
END_VAR

// Must be 0. Anything else means a failed fixture was treated as a working one.
PROPERTY BodyCalls : UDINT
GET
BodyCalls := _BodyCalls;
END_GET
END_PROPERTY

METHOD Run : BOOL
VAR_INPUT
	Enable : BOOL;
	Test   : I_TestAssertions;
END_VAR
IF Enable THEN
	_BodyCalls := _BodyCalls + 1;
	Test.AssertTrue(TRUE, 'the body should never reach this');
END_IF

Run := TRUE;
END_METHOD

METHOD Setup : BOOL
VAR_INPUT
	Enable : BOOL;
	Test   : I_TestAssertions;
END_VAR
Test.Fail('the fixture could not be brought up');
Setup := TRUE;
END_METHOD

METHOD Teardown : BOOL
VAR_INPUT
	Enable : BOOL;
	Test   : I_TestAssertions;
END_VAR
_TeardownCalls := _TeardownCalls + 1;
Teardown	   := TRUE;
END_METHOD

// Must be 1. Teardown is guaranteed whatever the verdict.
PROPERTY TeardownCalls : UDINT
GET
TeardownCalls := _TeardownCalls;
END_GET
END_PROPERTY

END_FUNCTION_BLOCK

// ---- Tests/Runner/TEST_RunnerSetupDoesNotSpendTheBodyBudget.TcPOU
// Setup can legitimately be slow. It must not spend the body's scan budget doing

// it, or a fixture waiting on hardware would time out work that never started.

//

// A body budget of ONE, and a setup taking four scans. If the two shared a clock

// this test would report a timeout instead of a pass.
FUNCTION_BLOCK TEST_RunnerSetupDoesNotSpendTheBodyBudget IMPLEMENTS I_Test
VAR
	// A private runner, driven one scan per call. The outer test spans scans by

	// returning FALSE, which is exactly the mechanism being verified one level down.
	Registry	   : TestRegistry<1>;
	Runner		   : TestRunner;
	Handle		   : TestVerdict;
	Budgets		   : ST_TestBudgets;
	Journal		   : REFERENCE TO TestJournal;
	Slot		   : ST_TestSlot;
	Outcome		   : E_PhaseOutcome;
	Loaded		   : BOOL;
	Phase		   : DINT;
	Scans		   : DINT;
	Subject		   : SlowSetupTest;
	ExpectedZero   : UDINT;
	ExpectedFour   : UDINT;
	ExpectedOne	   : UDINT;
	ActualCount	   : UDINT;
	ExpectedStatus : E_TestStatus;
	ActualStatus   : E_TestStatus;
END_VAR

METHOD Run : BOOL
VAR_INPUT
	Enable : BOOL;
	Test   : I_TestAssertions;
END_VAR
Scans := Scans + 1;
IF Scans > 200 THEN
	Test.Fail('the subject never reached a terminal outcome');
	Run := TRUE;
	RETURN;
END_IF

CASE Phase OF
	0:
		// One scan for the body. Four for setup, from the suite default, which is
		// deliberately left disabled here so setup cannot expire.
		Budgets.Body.Cycles		 := 1;
		Budgets.Body.IsCyclesSet := TRUE;
		Registry.TryClaim(Subject, 'slow setup', Budgets);
		Runner.Attach(Roster := Registry, Verdict := Handle);
		Slot   := Registry.Slot(0);
		Loaded := Runner.Load(Slot);
		Phase  := 1;
		Run	   := FALSE;

	1:
		Outcome := Runner.Advance(Enable := TRUE);
		IF Outcome <> E_PhaseOutcome.Running THEN
			Phase := 2;
		END_IF

		Run := FALSE;

	2:
		ExpectedFour := 4;
		ActualCount	 := Subject.SetupCalls;
		Test.AssertEqual(ExpectedFour, ActualCount, 'setup took four scans');
		ExpectedOne := 1;
		ActualCount := Subject.BodyCalls;
		Test.AssertEqual(ExpectedOne, ActualCount, 'the body still got its scan');

		// The proof: had setup spent the body budget, this would be four.
		ExpectedZero := 0;
		ActualCount	 := Subject.CyclesAtStart;
		Test.AssertEqual(ExpectedZero, ActualCount, 'the body started at zero cycles');
		Test.AssertTrue(Subject.FirstCycleAtStart, 'and its first call was the first cycle');
		Journal REF= Registry.Journal(0);
		IF __ISVALIDREF(Journal) THEN
			ExpectedStatus := E_TestStatus.Passed;
			ActualStatus   := Journal.Status;
			Test.AssertEqual(ExpectedStatus, ActualStatus, 'passed, not timed out');
		END_IF

		Run := TRUE;
END_CASE
END_METHOD

END_FUNCTION_BLOCK

// ---- Doubles/SlowSetupTest.TcPOU
// Setup that legitimately takes several scans - waiting for hardware to answer is

// the normal case, which is why setup has its own deadline.

//

// The body then records what the runner told it about timing. Setup must NOT have

// spent the body's scan budget, and the body's first call must still be its first

// cycle.
FUNCTION_BLOCK SlowSetupTest IMPLEMENTS I_Test, I_TestSetup
VAR
	_SetupScans		   : UDINT := 4;
	_SetupCalls		   : UDINT;
	_BodyCalls		   : UDINT;
	_FirstCycleAtStart : BOOL;
	_CyclesAtStart	   : UDINT;
END_VAR

PROPERTY BodyCalls : UDINT
GET
BodyCalls := _BodyCalls;
END_GET
END_PROPERTY

// ElapsedCycles as the body saw it on its first call. Zero if setup did not spend

// the body's budget.
PROPERTY CyclesAtStart : UDINT
GET
CyclesAtStart := _CyclesAtStart;
END_GET
END_PROPERTY

// TRUE if the body's first scan was reported as the first cycle, despite setup

// having consumed four scans before it.
PROPERTY FirstCycleAtStart : BOOL
GET
FirstCycleAtStart := _FirstCycleAtStart;
END_GET
END_PROPERTY

METHOD Run : BOOL
VAR_INPUT
	Enable : BOOL;
	Test   : I_TestAssertions;
END_VAR
IF NOT Enable THEN
	Run := TRUE;
	RETURN;
END_IF

_BodyCalls := _BodyCalls + 1;
IF _BodyCalls = 1 THEN
	_FirstCycleAtStart := Test.IsFirstCycle;
	_CyclesAtStart	   := Test.ElapsedCycles;
END_IF

Test.AssertTrue(TRUE, 'body ran after a slow setup');
Run := TRUE;
END_METHOD

METHOD Setup : BOOL
VAR_INPUT
	Enable : BOOL;
	Test   : I_TestAssertions;
END_VAR
IF NOT Enable THEN
	Setup := TRUE;
	RETURN;
END_IF

_SetupCalls := _SetupCalls + 1;
Setup		:= (_SetupCalls >= _SetupScans);
END_METHOD

PROPERTY SetupCalls : UDINT
GET
SetupCalls := _SetupCalls;
END_GET
END_PROPERTY

END_FUNCTION_BLOCK

// ---- Tests/Runner/TEST_RunnerBodyDeadlineFires.TcPOU
// A body that never finishes is stopped by its deadline rather than stalling the

// suite. Teardown is not implemented by this subject, so the runner must finish

// without one.
FUNCTION_BLOCK TEST_RunnerBodyDeadlineFires IMPLEMENTS I_Test
VAR
	// A private runner, driven one scan per call. The outer test spans scans by

	// returning FALSE, which is exactly the mechanism being verified one level down.
	Registry	   : TestRegistry<1>;
	Runner		   : TestRunner;
	Handle		   : TestVerdict;
	Budgets		   : ST_TestBudgets;
	Journal		   : REFERENCE TO TestJournal;
	Slot		   : ST_TestSlot;
	Outcome		   : E_PhaseOutcome;
	Loaded		   : BOOL;
	Phase		   : DINT;
	Scans		   : DINT;
	Subject		   : HangingBodyTest;
	ExpectedCycles : UDINT;
	ActualCycles   : UDINT;
	ExpectedKind   : E_FailureKind;
	ActualKind	   : E_FailureKind;
	ExpectedStatus : E_TestStatus;
	ActualStatus   : E_TestStatus;
END_VAR

METHOD Run : BOOL
VAR_INPUT
	Enable : BOOL;
	Test   : I_TestAssertions;
END_VAR
Scans := Scans + 1;
IF Scans > 200 THEN
	Test.Fail('the subject never reached a terminal outcome');
	Run := TRUE;
	RETURN;
END_IF

CASE Phase OF
	0:
		Budgets.Body.Cycles		 := 3;
		Budgets.Body.IsCyclesSet := TRUE;
		Registry.TryClaim(Subject, 'hangs', Budgets);
		Runner.Attach(Roster := Registry, Verdict := Handle);
		Slot   := Registry.Slot(0);
		Loaded := Runner.Load(Slot);
		Phase  := 1;
		Run	   := FALSE;

	1:
		Outcome := Runner.Advance(Enable := TRUE);
		IF Outcome <> E_PhaseOutcome.Running THEN
			Phase := 2;
		END_IF

		Run := FALSE;

	2:
		Test.AssertTrue(Outcome = E_PhaseOutcome.Finished, 'the runner finished it');
		ExpectedCycles := 3;
		ActualCycles   := Subject.BodyCalls;
		Test.AssertEqual(ExpectedCycles, ActualCycles, 'the body got its whole budget');
		Journal REF= Registry.Journal(0);
		IF __ISVALIDREF(Journal) THEN
			ExpectedKind := E_FailureKind.Timeout;
			ActualKind	 := Journal.Kind;
			Test.AssertEqual(ExpectedKind, ActualKind, 'recorded as a timeout');
			ExpectedStatus := E_TestStatus.Failed;
			ActualStatus   := Journal.Status;
			Test.AssertEqual(ExpectedStatus, ActualStatus, 'and Failed');
		END_IF

		Run := TRUE;
END_CASE
END_METHOD

END_FUNCTION_BLOCK

// ---- Doubles/HangingBodyTest.TcPOU
// A body that never finishes. The deadline must stop it - this is the failure

// mode the whole timeout mechanism exists for.

//

// Also counts the abandon call, because a hung test is exactly the one that will

// not answer a falling Enable either. The runner makes ONE such call and ignores

// the return.
FUNCTION_BLOCK HangingBodyTest IMPLEMENTS I_Test
VAR
	_BodyCalls	  : UDINT;
	_AbandonCalls : UDINT;
END_VAR

